   1:  PR[GP1:91,2] = PR[GP1:90,2] + 93.365;
   1:L PR[91] 10mm/sec FINE;
   1:  PR[GP1:91,1] = PR[GP1:90,1] + 106.411;
   1:  PR[GP1:91,2] = PR[GP1:90,2] + 92.968;
   1:L PR[91] 10mm/sec FINE;
   1:  PR[GP1:91,1] = PR[GP1:90,1] + 107.868;
   1:  PR[GP1:91,2] = PR[GP1:90,2] + 92.513;
   1:L PR[91] 10mm/sec FINE;
   1:  PR[GP1:91,1] = PR[GP1:90,1] + 110.644;
   1:  PR[GP1:91,2] = PR[GP1:90,2] + 92.029;
   1:L PR[91] 10mm/sec FINE;
   1:  PR[GP1:91,1] = PR[GP1:90,1] + 113.585;
   1:  PR[GP1:91,2] = PR[GP1:90,2] + 91.917;
   1:L PR[91] 10mm/sec FINE;
   1:  PR[GP1:91,1] = PR[GP1:90,1] + 116.531;
   1:  PR[GP1:91,2] = PR[GP1:90,2] + 92.230;
   1:L PR[91] 10mm/sec FINE;
   1:  PR[GP1:91,1] = PR[GP1:90,1] + 119.377;
   1:  PR[GP1:91,2] = PR[GP1:90,2] + 92.959;
   1:L PR[91] 10mm/sec FINE;
   1:  PR[GP1:91,1] = PR[GP1:90,1] + 121.994;
   1:  PR[GP1:91,2] = PR[GP1:90,2] + 94.064;
   1:L PR[91] 10mm/sec FINE;
   1:  PR[GP1:91,1] = PR[GP1:90,1] + 124.401;
   1:  PR[GP1:91,2] = PR[GP1:90,2] + 95.539;
   1:L PR[91] 10mm/sec FINE;
   1:  PR[GP1:91,1] = PR[GP1:90,1] + 126.542;
   1:  PR[GP1:91,2] = PR[GP1:90,2] + 97.347;
   1:L PR[91] 10mm/sec FINE;
   1:  PR[GP1:91,1] = PR[GP1:90,1] + 128.367;
   1:  PR[GP1:91,2] = PR[GP1:90,2] + 99.443;
   1:L PR[91] 10mm/sec FINE;
   1:  PR[GP1:91,1] = PR[GP1:90,1] + 129.834;
   1:  PR[GP1:91,2] = PR[GP1:90,2] + 101.778;
   1:L PR[91] 10mm/sec FINE;
   1:  PR[GP1:91,1] = PR[GP1:90,1] + 130.082;
   1:  PR[GP1:91,2] = PR[GP1:90,2] + 102.358;
   1:L PR[91] 10mm/sec FINE;
   1:  PR[GP1:91,1] = PR[GP1:90,1] + 130.881;
   1:  PR[GP1:91,2] = PR[GP1:90,2] + 104.290;
   1:L PR[91] 10mm/sec FINE;
   1:  PR[GP1:91,1] = PR[GP1:90,1] + 131.513;
   1:  PR[GP1:91,2] = PR[GP1:90,2] + 106.930;
   1:L PR[91] 10mm/sec FINE;
   1:  PR[GP1:91,1] = PR[GP1:90,1] + 131.608;
   1:  PR[GP1:91,2] = PR[GP1:90,2] + 107.870;
   1:L PR[91] 10mm/sec FINE;
   1:  PR[GP1:91,1] = PR[GP1:90,1] + 131.746;
   1:  PR[GP1:91,2] = PR[GP1:90,2] + 109.629;
   1:L PR[91] 10mm/sec FINE;
   1:  PR[GP1:91,1] = PR[GP1:90,1] + 131.403;
   1:  PR[GP1:91,2] = PR[GP1:90,2] + 113.038;
   1:L PR[91] 10mm/sec FINE;
   1:  PR[GP1:91,1] = PR[GP1:90,1] + 130.376;
   1:  PR[GP1:91,2] = PR[GP1:90,2] + 116.309;
   1:L PR[91] 10mm/sec FINE;
   1:  PR[GP1:91,1] = PR[GP1:90,1] + 128.692;
   1:  PR[GP1:91,2] = PR[GP1:90,2] + 119.314;
   1:L PR[91] 10mm/sec FINE;
   1:  PR[GP1:91,1] = PR[GP1:90,1] + 126.422;
   1:  PR[GP1:91,2] = PR[GP1:90,2] + 121.938;
   1:L PR[91] 10mm/sec FINE;
   1:  PR[GP1:91,1] = PR[GP1:90,1] + 123.656;
   1:  PR[GP1:91,2] = PR[GP1:90,2] + 124.077;
   1:L PR[91] 10mm/sec FINE;
   1:  PR[GP1:91,1] = PR[GP1:90,1] + 120.503;
   1:  PR[GP1:91,2] = PR[GP1:90,2] + 125.648;
   1:L PR[91] 10mm/sec FINE;
   1:  PR[GP1:91,1] = PR[GP1:90,1] + 117.094;
   1:  PR[GP1:91,2] = PR[GP1:90,2] + 126.591;
   1:L PR[91] 10mm/sec FINE;
   1:  PR[GP1:91,1] = PR[GP1:90,1] + 113.460;
   1:  PR[GP1:91,2] = PR[GP1:90,2] + 126.855;
   1:L PR[91] 10mm/sec FINE;
   1:  PR[GP1:91,1] = PR[GP1:90,1] + 109.815;
   1:  PR[GP1:91,2] = PR[GP1:90,2] + 126.442;
   1:L PR[91] 10mm/sec FINE;
   1:  PR[GP1:91,1] = PR[GP1:90,1] + 106.259;
   1:  PR[GP1:91,2] = PR[GP1:90,2] + 125.353;
   1:L PR[91] 10mm/sec FINE;
   1:  PR[GP1:91,1] = PR[GP1:90,1] + 102.967;
   1:  PR[GP1:91,2] = PR[GP1:90,2] + 123.644;
   1:L PR[91] 10mm/sec FINE;
   1:  PR[GP1:91,1] = PR[GP1:90,1] + 100.053;
   1:  PR[GP1:91,2] = PR[GP1:90,2] + 121.370;
   1:L PR[91] 10mm/sec FINE;
   1:  PR[GP1:91,1] = PR[GP1:90,1] + 97.658;
   1:  PR[GP1:91,2] = PR[GP1:90,2] + 118.630;
   1:L PR[91] 10mm/sec FINE;
   1:  PR[GP1:91,1] = PR[GP1:90,1] + 97.573;
   1:  PR[GP1:91,2] = PR[GP1:90,2] + 118.506;
   1:L PR[91] 10mm/sec FINE;
   1:  PR[GP1:91,1] = PR[GP1:90,1] + 96.390;
   1:  PR[GP1:91,2] = PR[GP1:90,2] + 116.490;
   1:L PR[91] 10mm/sec FINE;
   1:  PR[GP1:91,1] = PR[GP1:90,1] + 96.144;
   1:  PR[GP1:91,2] = PR[GP1:90,2] + 116.224;
   1:L PR[91] 10mm/sec FINE;
   1:  PR[GP1:91,1] = PR[GP1:90,1] + 95.665;
   1:  PR[GP1:91,2] = PR[GP1:90,2] + 115.648;
   1:L PR[91] 10mm/sec FINE;
   1:  PR[GP1:91,1] = PR[GP1:90,1] + 94.894;
   1:  PR[GP1:91,2] = PR[GP1:90,2] + 115.385;
   1:L PR[91] 10mm/sec FINE;
   1:  PR[GP1:91,1] = PR[GP1:90,1] + 94.595;
   1:  PR[GP1:91,2] = PR[GP1:90,2] + 115.322;
   1:L PR[91] 10mm/sec FINE;
   1:  PR[GP1:91,1] = PR[GP1:90,1] + 94.212;
   1:  PR[GP1:91,2] = PR[GP1:90,2] + 115.485;
   1:L PR[91] 10mm/sec FINE;
   1:  PR[GP1:91,1] = PR[GP1:90,1] + 93.542;
   1:  PR[GP1:91,2] = PR[GP1:90,2] + 115.632;
   1:L PR[91] 10mm/sec FINE;
   1:  PR[GP1:91,1] = PR[GP1:90,1] + 92.998;
   1:  PR[GP1:91,2] = PR[GP1:90,2] + 116.268;
   1:L PR[91] 10mm/sec FINE;
   1:  PR[GP1:91,1] = PR[GP1:90,1] + 92.725;
   1:  PR[GP1:91,2] = PR[GP1:90,2] + 116.535;
   1:L PR[91] 10mm/sec FINE;
   1:  PR[GP1:91,1] = PR[GP1:90,1] + 92.039;
   1:  PR[GP1:91,2] = PR[GP1:90,2] + 117.892;
   1:L PR[91] 10mm/sec FINE;
   1:  PR[GP1:91,1] = PR[GP1:90,1] + 91.114;
   1:  PR[GP1:91,2] = PR[GP1:90,2] + 119.148;
   1:L PR[91] 10mm/sec FINE;
   1:  PR[GP1:91,1] = PR[GP1:90,1] + 89.807;
   1:  PR[GP1:91,2] = PR[GP1:90,2] + 120.838;
   1:L PR[91] 10mm/sec FINE;
   1:  PR[GP1:91,1] = PR[GP1:90,1] + 89.143;
   1:  PR[GP1:91,2] = PR[GP1:90,2] + 121.442;
   1:L PR[91] 10mm/sec FINE;
   1:  PR[GP1:91,1] = PR[GP1:90,1] + 87.033;
   1:  PR[GP1:91,2] = PR[GP1:90,2] + 123.279;
   1:L PR[91] 10mm/sec FINE;
   1:  PR[GP1:91,1] = PR[GP1:90,1] + 84.036;
   1:  PR[GP1:91,2] = PR[GP1:90,2] + 125.037;
   1:L PR[91] 10mm/sec FINE;
   1:  PR[GP1:91,1] = PR[GP1:90,1] + 83.776;
   1:  PR[GP1:91,2] = PR[GP1:90,2] + 125.157;
   1:L PR[91] 10mm/sec FINE;
   1:  PR[GP1:91,1] = PR[GP1:90,1] + 80.948;
   1:  PR[GP1:91,2] = PR[GP1:90,2] + 126.151;
   1:L PR[91] 10mm/sec FINE;
   1:  PR[GP1:91,1] = PR[GP1:90,1] + 80.100;
   1:  PR[GP1:91,2] = PR[GP1:90,2] + 126.346;
   1:L PR[91] 10mm/sec FINE;
   1:  PR[GP1:91,1] = PR[GP1:90,1] + 77.624;
   1:  PR[GP1:91,2] = PR[GP1:90,2] + 126.695;
   1:L PR[91] 10mm/sec FINE;
   1:  PR[GP1:91,1] = PR[GP1:90,1] + 76.257;
   1:  PR[GP1:91,2] = PR[GP1:90,2] + 126.719;
   1:L PR[91] 10mm/sec FINE;
   1:  PR[GP1:91,1] = PR[GP1:90,1] + 74.185;
   1:  PR[GP1:91,2] = PR[GP1:90,2] + 126.597;
   1:L PR[91] 10mm/sec FINE;
   1:  PR[GP1:91,1] = PR[GP1:90,1] + 72.443;
   1:  PR[GP1:91,2] = PR[GP1:90,2] + 126.260;
   1:L PR[91] 10mm/sec FINE;
   1:  PR[GP1:91,1] = PR[GP1:90,1] + 70.778;
   1:  PR[GP1:91,2] = PR[GP1:90,2] + 125.820;
   1:L PR[91] 10mm/sec FINE;
   1:  PR[GP1:91,1] = PR[GP1:90,1] + 68.849;
   1:  PR[GP1:91,2] = PR[GP1:90,2] + 125.002;
   1:L PR[91] 10mm/sec FINE;
   1:  PR[GP1:91,1] = PR[GP1:90,1] + 67.556;
   1:  PR[GP1:91,2] = PR[GP1:90,2] + 124.364;
   1:L PR[91] 10mm/sec FINE;
   1:  PR[GP1:91,1] = PR[GP1:90,1] + 65.645;
   1:  PR[GP1:91,2] = PR[GP1:90,2] + 123.022;
   1:L PR[91] 10mm/sec FINE;
   1:  PR[GP1:91,1] = PR[GP1:90,1] + 64.673;
   1:  PR[GP1:91,2] = PR[GP1:90,2] + 122.267;
   1:L PR[91] 10mm/sec FINE;
   1:  PR[GP1:91,1] = PR[GP1:90,1] + 62.978;
   1:  PR[GP1:91,2] = PR[GP1:90,2] + 120.431;
   1:L PR[91] 10mm/sec FINE;
   1:  PR[GP1:91,1] = PR[GP1:90,1] + 62.273;
   1:  PR[GP1:91,2] = PR[GP1:90,2] + 119.605;
   1:L PR[91] 10mm/sec FINE;
   1:  PR[GP1:91,1] = PR[GP1:90,1] + 60.958;
   1:  PR[GP1:91,2] = PR[GP1:90,2] + 117.370;
   1:L PR[91] 10mm/sec FINE;
   1:  PR[GP1:91,1] = PR[GP1:90,1] + 60.473;
   1:  PR[GP1:91,2] = PR[GP1:90,2] + 116.491;
   1:L PR[91] 10mm/sec FINE;
   1:  PR[GP1:91,1] = PR[GP1:90,1] + 59.651;
   1:  PR[GP1:91,2] = PR[GP1:90,2] + 113.998;
   1:L PR[91] 10mm/sec FINE;
   1:  PR[GP1:91,1] = PR[GP1:90,1] + 59.357;
   1:  PR[GP1:91,2] = PR[GP1:90,2] + 113.064;
   1:L PR[91] 10mm/sec FINE;
   1:  PR[GP1:91,1] = PR[GP1:90,1] + 59.093;
   1:  PR[GP1:91,2] = PR[GP1:90,2] + 110.477;
   1:L PR[91] 10mm/sec FINE;
   1:  PR[GP1:91,1] = PR[GP1:90,1] + 58.933;
   1:  PR[GP1:91,2] = PR[GP1:90,2] + 109.489;
   1:L PR[91] 10mm/sec FINE;
   1:  PR[GP1:91,1] = PR[GP1:90,1] + 59.068;
   1:  PR[GP1:91,2] = PR[GP1:90,2] + 108.273;
   1:L PR[91] 10mm/sec FINE;
   1:  PR[GP1:91,1] = PR[GP1:90,1] + 59.281;
   1:  PR[GP1:91,2] = PR[GP1:90,2] + 106.982;
   1:L PR[91] 10mm/sec FINE;
   1:  PR[GP1:91,1] = PR[GP1:90,1] + 59.404;
   1:  PR[GP1:91,2] = PR[GP1:90,2] + 105.878;
   1:L PR[91] 10mm/sec FINE;
   1:  PR[GP1:91,1] = PR[GP1:90,1] + 59.777;
   1:  PR[GP1:91,2] = PR[GP1:90,2] + 104.702;
   1:L PR[91] 10mm/sec FINE;
   1:  PR[GP1:91,1] = PR[GP1:90,1] + 60.530;
   1:  PR[GP1:91,2] = PR[GP1:90,2] + 102.461;
   1:L PR[91] 10mm/sec FINE;
   1:  PR[GP1:91,1] = PR[GP1:90,1] + 61.244;
   1:  PR[GP1:91,2] = PR[GP1:90,2] + 101.193;
   1:L PR[91] 10mm/sec FINE;
   1:  PR[GP1:91,1] = PR[GP1:90,1] + 62.336;
   1:  PR[GP1:91,2] = PR[GP1:90,2] + 99.359;
   1:L PR[91] 10mm/sec FINE;
   1:  PR[GP1:91,1] = PR[GP1:90,1] + 63.483;
   1:  PR[GP1:91,2] = PR[GP1:90,2] + 98.037;
   1:L PR[91] 10mm/sec FINE;
   1:  PR[GP1:91,1] = PR[GP1:90,1] + 64.717;
   1:  PR[GP1:91,2] = PR[GP1:90,2] + 96.705;
   1:L PR[91] 10mm/sec FINE;
   1:  PR[GP1:91,1] = PR[GP1:90,1] + 66.397;
   1:  PR[GP1:91,2] = PR[GP1:90,2] + 95.413;
   1:L PR[91] 10mm/sec FINE;
   1:  PR[GP1:91,1] = PR[GP1:90,1] + 67.544;
   1:  PR[GP1:91,2] = PR[GP1:90,2] + 94.604;
   1:L PR[91] 10mm/sec FINE;
   1:  PR[GP1:91,1] = PR[GP1:90,1] + 70.520;
   1:  PR[GP1:91,2] = PR[GP1:90,2] + 93.186;
   1:  PR[GP1:91,3] = PR[GP1:90,3] + 14.900;
   1:L PR[91] 10mm/sec FINE;
   1:  PR[GP1:91,1] = PR[GP1:90,1] + 70.665;
   1:  PR[GP1:91,2] = PR[GP1:90,2] + 93.124;
   1:L PR[91] 10mm/sec FINE;
   1:  PR[GP1:91,1] = PR[GP1:90,1] + 74.193;
   1:  PR[GP1:91,2] = PR[GP1:90,2] + 92.191;
   1:L PR[91] 10mm/sec FINE;
   1:  PR[GP1:91,1] = PR[GP1:90,1] + 76.941;
   1:  PR[GP1:91,2] = PR[GP1:90,2] + 91.997;
   1:L PR[91] 10mm/sec FINE;
   1:  PR[GP1:91,1] = PR[GP1:90,1] + 77.958;
   1:  PR[GP1:91,2] = PR[GP1:90,2] + 91.958;
   1:L PR[91] 10mm/sec FINE;
   1:  PR[GP1:91,1] = PR[GP1:90,1] + 80.017;
   1:  PR[GP1:91,2] = PR[GP1:90,2] + 92.214;
   1:L PR[91] 10mm/sec FINE;
   1:  PR[GP1:91,1] = PR[GP1:90,1] + 81.716;
   1:  PR[GP1:91,2] = PR[GP1:90,2] + 92.489;
   1:L PR[91] 10mm/sec FINE;
   1:  PR[GP1:91,1] = PR[GP1:90,1] + 82.974;
   1:  PR[GP1:91,2] = PR[GP1:90,2] + 92.908;
   1:L PR[91] 10mm/sec FINE;
   1:  PR[GP1:91,1] = PR[GP1:90,1] + 85.293;
   1:  PR[GP1:91,2] = PR[GP1:90,2] + 93.785;
   1:L PR[91] 10mm/sec FINE;
   1:  PR[GP1:91,1] = PR[GP1:90,1] + 85.763;
   1:  PR[GP1:91,2] = PR[GP1:90,2] + 94.055;
   1:L PR[91] 10mm/sec FINE;
   1:  PR[GP1:91,1] = PR[GP1:90,1] + 87.717;
   1:  PR[GP1:91,2] = PR[GP1:90,2] + 95.298;
   1:L PR[91] 10mm/sec FINE;
   1:  PR[GP1:91,1] = PR[GP1:90,1] + 88.397;
   1:  PR[GP1:91,2] = PR[GP1:90,2] + 95.701;
   1:L PR[91] 10mm/sec FINE;
   1:  PR[GP1:91,1] = PR[GP1:90,1] + 88.557;
   1:  PR[GP1:91,2] = PR[GP1:90,2] + 95.813;
   1:L PR[91] 10mm/sec FINE;
   1:  PR[GP1:91,1] = PR[GP1:90,1] + 90.767;
   1:  PR[GP1:91,2] = PR[GP1:90,2] + 97.865;
   1:L PR[91] 10mm/sec FINE;
   1:  PR[GP1:91,1] = PR[GP1:90,1] + 91.387;
   1:  PR[GP1:91,2] = PR[GP1:90,2] + 98.554;
   1:L PR[91] 10mm/sec FINE;
   1:  PR[GP1:91,1] = PR[GP1:90,1] + 92.812;
   1:  PR[GP1:91,2] = PR[GP1:90,2] + 100.657;
   1:L PR[91] 10mm/sec FINE;
   1:  PR[GP1:91,1] = PR[GP1:90,1] + 93.383;
   1:  PR[GP1:91,2] = PR[GP1:90,2] + 101.249;
   1:L PR[91] 10mm/sec FINE;
   1:  PR[GP1:91,1] = PR[GP1:90,1] + 93.641;
   1:  PR[GP1:91,2] = PR[GP1:90,2] + 101.422;
   1:L PR[91] 10mm/sec FINE;
   1:  PR[GP1:91,1] = PR[GP1:90,1] + 94.275;
   1:  PR[GP1:91,2] = PR[GP1:90,2] + 101.612;
   1:L PR[91] 10mm/sec FINE;
   1:  PR[GP1:91,1] = PR[GP1:90,1] + 94.605;
   1:  PR[GP1:91,2] = PR[GP1:90,2] + 101.633;
   1:L PR[91] 10mm/sec FINE;
   1:  PR[GP1:91,1] = PR[GP1:90,1] + 95.231;
   1:  PR[GP1:91,2] = PR[GP1:90,2] + 101.437;
   1:L PR[91] 10mm/sec FINE;
   1:  PR[GP1:91,1] = PR[GP1:90,1] + 95.508;
   1:  PR[GP1:91,2] = PR[GP1:90,2] + 101.289;
   1:L PR[91] 10mm/sec FINE;
   1:  PR[GP1:91,1] = PR[GP1:90,1] + 96.060;
   1:  PR[GP1:91,2] = PR[GP1:90,2] + 100.681;
   1:L PR[91] 10mm/sec FINE;
   1:  PR[GP1:91,1] = PR[GP1:90,1] + 96.158;
   1:  PR[GP1:91,2] = PR[GP1:90,2] + 100.460;
   1:L PR[91] 10mm/sec FINE;
   1:  PR[GP1:91,1] = PR[GP1:90,1] + 96.407;
   1:  PR[GP1:91,2] = PR[GP1:90,2] + 100.056;
   1:L PR[91] 10mm/sec FINE;
   1:  PR[GP1:91,1] = PR[GP1:90,1] + 97.376;
   1:  PR[GP1:91,2] = PR[GP1:90,2] + 98.732;
   1:L PR[91] 10mm/sec FINE;
   1:  PR[GP1:91,1] = PR[GP1:90,1] + 98.317;
   1:  PR[GP1:91,2] = PR[GP1:90,2] + 97.605;
   1:L PR[91] 10mm/sec FINE;
   1:  PR[GP1:91,1] = PR[GP1:90,1] + 99.415;
   1:  PR[GP1:91,2] = PR[GP1:90,2] + 96.557;
   1:L PR[91] 10mm/sec FINE;
   1:  PR[GP1:91,1] = PR[GP1:90,1] + 100.269;
   1:  PR[GP1:91,2] = PR[GP1:90,2] + 95.816;
   1:L PR[91] 10mm/sec FINE;
   1:  PR[GP1:91,1] = PR[GP1:90,1] + 101.945;
   1:  PR[GP1:91,2] = PR[GP1:90,2] + 94.671;
   1:L PR[91] 10mm/sec FINE;
   1:  PR[GP1:91,1] = PR[GP1:90,1] + 102.489;
   1:  PR[GP1:91,2] = PR[GP1:90,2] + 94.332;
   1:L PR[91] 10mm/sec FINE;
   1:  PR[GP1:91,1] = PR[GP1:90,1] + 104.935;
   1:  PR[GP1:91,2] = PR[GP1:90,2] + 93.175;
   1:L PR[91] 10mm/sec FINE;
   1:  PR[GP1:91,1] = PR[GP1:90,1] + 107.578;
   1:  PR[GP1:91,2] = PR[GP1:90,2] + 92.350;
   1:L PR[91] 10mm/sec FINE;
   1:  PR[GP1:91,1] = PR[GP1:90,1] + 108.827;
   1:  PR[GP1:91,2] = PR[GP1:90,2] + 92.129;
   1:L PR[91] 10mm/sec FINE;
   1:  PR[GP1:91,1] = PR[GP1:90,1] + 110.348;
   1:  PR[GP1:91,2] = PR[GP1:90,2] + 91.892;
   1:L PR[91] 10mm/sec FINE;
   1:  PR[GP1:91,1] = PR[GP1:90,1] + 113.198;
   1:  PR[GP1:91,2] = PR[GP1:90,2] + 91.815;
   1:L PR[91] 10mm/sec FINE;
   1:  PR[GP1:91,1] = PR[GP1:90,1] + 116.141;
   1:  PR[GP1:91,2] = PR[GP1:90,2] + 92.132;
   1:L PR[91] 10mm/sec FINE;
   1:  PR[GP1:91,1] = PR[GP1:90,1] + 119.006;
   1:  PR[GP1:91,2] = PR[GP1:90,2] + 92.868;
   1:L PR[91] 10mm/sec FINE;
   1:  PR[GP1:91,1] = PR[GP1:90,1] + 121.709;
   1:  PR[GP1:91,2] = PR[GP1:90,2] + 94.002;
   1:L PR[91] 10mm/sec FINE;
   1:  PR[GP1:91,1] = PR[GP1:90,1] + 124.119;
   1:  PR[GP1:91,2] = PR[GP1:90,2] + 95.482;
   1:L PR[91] 10mm/sec FINE;
   1:  PR[GP1:91,1] = PR[GP1:90,1] + 126.262;
   1:  PR[GP1:91,2] = PR[GP1:90,2] + 97.295;
   1:L PR[91] 10mm/sec FINE;
   1:  PR[GP1:91,1] = PR[GP1:90,1] + 128.087;
   1:  PR[GP1:91,2] = PR[GP1:90,2] + 99.396;
   1:L PR[91] 10mm/sec FINE;
   1:  PR[GP1:91,1] = PR[GP1:90,1] + 129.553;
   1:  PR[GP1:91,2] = PR[GP1:90,2] + 101.737;
   1:L PR[91] 10mm/sec FINE;
   1:  PR[GP1:91,1] = PR[GP1:90,1] + 130.628;
   1:  PR[GP1:91,2] = PR[GP1:90,2] + 104.259;
   1:L PR[91] 10mm/sec FINE;
   1:  PR[GP1:91,1] = PR[GP1:90,1] + 131.284;
   1:  PR[GP1:91,2] = PR[GP1:90,2] + 106.903;
   1:L PR[91] 10mm/sec FINE;
   1:  PR[GP1:91,1] = PR[GP1:90,1] + 131.512;
   1:  PR[GP1:91,2] = PR[GP1:90,2] + 109.606;
   1:L PR[91] 10mm/sec FINE;
   1:  PR[GP1:91,1] = PR[GP1:90,1] + 131.132;
   1:  PR[GP1:91,2] = PR[GP1:90,2] + 113.012;
   1:L PR[91] 10mm/sec FINE;
   1:  PR[GP1:91,1] = PR[GP1:90,1] + 130.096;
   1:  PR[GP1:91,2] = PR[GP1:90,2] + 116.285;
   1:L PR[91] 10mm/sec FINE;
   1:  PR[GP1:91,1] = PR[GP1:90,1] + 128.408;
   1:  PR[GP1:91,2] = PR[GP1:90,2] + 119.291;
   1:L PR[91] 10mm/sec FINE;
   1:  PR[GP1:91,1] = PR[GP1:90,1] + 126.135;
   1:  PR[GP1:91,2] = PR[GP1:90,2] + 121.914;
   1:L PR[91] 10mm/sec FINE;
   1:  PR[GP1:91,1] = PR[GP1:90,1] + 123.367;
   1:  PR[GP1:91,2] = PR[GP1:90,2] + 124.053;
   1:L PR[91] 10mm/sec FINE;
   1:  PR[GP1:91,1] = PR[GP1:90,1] + 120.214;
   1:  PR[GP1:91,2] = PR[GP1:90,2] + 125.623;
   1:L PR[91] 10mm/sec FINE;
   1:  PR[GP1:91,1] = PR[GP1:90,1] + 116.723;
   1:  PR[GP1:91,2] = PR[GP1:90,2] + 126.554;
   1:L PR[91] 10mm/sec FINE;
   1:  PR[GP1:91,1] = PR[GP1:90,1] + 113.071;
   1:  PR[GP1:91,2] = PR[GP1:90,2] + 126.814;
   1:L PR[91] 10mm/sec FINE;
   1:  PR[GP1:91,1] = PR[GP1:90,1] + 110.735;
   1:  PR[GP1:91,2] = PR[GP1:90,2] + 126.549;
   1:L PR[91] 10mm/sec FINE;
   1:  PR[GP1:91,1] = PR[GP1:90,1] + 109.397;
   1:  PR[GP1:91,2] = PR[GP1:90,2] + 126.390;
   1:L PR[91] 10mm/sec FINE;
   1:  PR[GP1:91,1] = PR[GP1:90,1] + 105.817;
   1:  PR[GP1:91,2] = PR[GP1:90,2] + 125.295;
   1:L PR[91] 10mm/sec FINE;
   1:  PR[GP1:91,1] = PR[GP1:90,1] + 102.508;
   1:  PR[GP1:91,2] = PR[GP1:90,2] + 123.573;
   1:L PR[91] 10mm/sec FINE;
   1:  PR[GP1:91,1] = PR[GP1:90,1] + 99.591;
   1:  PR[GP1:91,2] = PR[GP1:90,2] + 121.302;
   1:L PR[91] 10mm/sec FINE;
   1:  PR[GP1:91,1] = PR[GP1:90,1] + 97.207;
   1:  PR[GP1:91,2] = PR[GP1:90,2] + 118.552;
   1:L PR[91] 10mm/sec FINE;
   1:  PR[GP1:91,1] = PR[GP1:90,1] + 96.820;
   1:  PR[GP1:91,2] = PR[GP1:90,2] + 117.991;
   1:L PR[91] 10mm/sec FINE;
   1:  PR[GP1:91,1] = PR[GP1:90,1] + 96.302;
   1:  PR[GP1:91,2] = PR[GP1:90,2] + 117.108;
   1:L PR[91] 10mm/sec FINE;
   1:  PR[GP1:91,1] = PR[GP1:90,1] + 95.879;
   1:  PR[GP1:91,2] = PR[GP1:90,2] + 116.651;
   1:L PR[91] 10mm/sec FINE;
   1:  PR[GP1:91,1] = PR[GP1:90,1] + 95.563;
   1:  PR[GP1:91,2] = PR[GP1:90,2] + 116.270;
   1:L PR[91] 10mm/sec FINE;
   1:  PR[GP1:91,1] = PR[GP1:90,1] + 95.048;
   1:  PR[GP1:91,2] = PR[GP1:90,2] + 116.094;
   1:L PR[91] 10mm/sec FINE;
   1:  PR[GP1:91,1] = PR[GP1:90,1] + 94.485;
   1:  PR[GP1:91,2] = PR[GP1:90,2] + 115.975;
   1:L PR[91] 10mm/sec FINE;
   1:  PR[GP1:91,1] = PR[GP1:90,1] + 93.699;
   1:  PR[GP1:91,2] = PR[GP1:90,2] + 116.310;
   1:L PR[91] 10mm/sec FINE;
   1:  PR[GP1:91,1] = PR[GP1:90,1] + 93.425;
   1:  PR[GP1:91,2] = PR[GP1:90,2] + 116.370;
   1:L PR[91] 10mm/sec FINE;
   1:  PR[GP1:91,1] = PR[GP1:90,1] + 92.649;
   1:  PR[GP1:91,2] = PR[GP1:90,2] + 117.254;
   1:L PR[91] 10mm/sec FINE;
   1:  PR[GP1:91,1] = PR[GP1:90,1] + 92.414;
   1:  PR[GP1:91,2] = PR[GP1:90,2] + 117.704;
   1:L PR[91] 10mm/sec FINE;
   1:  PR[GP1:91,1] = PR[GP1:90,1] + 90.988;
   1:  PR[GP1:91,2] = PR[GP1:90,2] + 119.641;
   1:L PR[91] 10mm/sec FINE;
   1:  PR[GP1:91,1] = PR[GP1:90,1] + 90.184;
   1:  PR[GP1:91,2] = PR[GP1:90,2] + 120.680;
   1:L PR[91] 10mm/sec FINE;
   1:  PR[GP1:91,1] = PR[GP1:90,1] + 88.950;
   1:  PR[GP1:91,2] = PR[GP1:90,2] + 121.803;
   1:L PR[91] 10mm/sec FINE;
   1:  PR[GP1:91,1] = PR[GP1:90,1] + 87.405;
   1:  PR[GP1:91,2] = PR[GP1:90,2] + 123.148;
   1:L PR[91] 10mm/sec FINE;
   1:  PR[GP1:91,1] = PR[GP1:90,1] + 86.560;
   1:  PR[GP1:91,2] = PR[GP1:90,2] + 123.657;
   1:L PR[91] 10mm/sec FINE;
   1:  PR[GP1:91,1] = PR[GP1:90,1] + 84.204;
   1:  PR[GP1:91,2] = PR[GP1:90,2] + 125.014;
   1:L PR[91] 10mm/sec FINE;
   1:  PR[GP1:91,1] = PR[GP1:90,1] + 80.822;
   1:  PR[GP1:91,2] = PR[GP1:90,2] + 126.190;
   1:L PR[91] 10mm/sec FINE;
   1:  PR[GP1:91,1] = PR[GP1:90,1] + 80.672;
   1:  PR[GP1:91,2] = PR[GP1:90,2] + 126.224;
   1:L PR[91] 10mm/sec FINE;
   1:  PR[GP1:91,1] = PR[GP1:90,1] + 77.538;
   1:  PR[GP1:91,2] = PR[GP1:90,2] + 126.665;
   1:L PR[91] 10mm/sec FINE;
   1:  PR[GP1:91,1] = PR[GP1:90,1] + 76.839;
   1:  PR[GP1:91,2] = PR[GP1:90,2] + 126.678;
   1:L PR[91] 10mm/sec FINE;
   1:  PR[GP1:91,1] = PR[GP1:90,1] + 74.147;
   1:  PR[GP1:91,2] = PR[GP1:90,2] + 126.520;
   1:L PR[91] 10mm/sec FINE;
   1:  PR[GP1:91,1] = PR[GP1:90,1] + 73.019;
   1:  PR[GP1:91,2] = PR[GP1:90,2] + 126.301;
   1:L PR[91] 10mm/sec FINE;
   1:  PR[GP1:91,1] = PR[GP1:90,1] + 70.787;
   1:  PR[GP1:91,2] = PR[GP1:90,2] + 125.712;
   1:L PR[91] 10mm/sec FINE;
   1:  PR[GP1:91,1] = PR[GP1:90,1] + 69.401;
   1:  PR[GP1:91,2] = PR[GP1:90,2] + 125.124;
   1:L PR[91] 10mm/sec FINE;
   1:  PR[GP1:91,1] = PR[GP1:90,1] + 67.609;
   1:  PR[GP1:91,2] = PR[GP1:90,2] + 124.240;
   1:L PR[91] 10mm/sec FINE;
   1:  PR[GP1:91,1] = PR[GP1:90,1] + 66.159;
   1:  PR[GP1:91,2] = PR[GP1:90,2] + 123.220;
   1:L PR[91] 10mm/sec FINE;
   1:  PR[GP1:91,1] = PR[GP1:90,1] + 64.767;
   1:  PR[GP1:91,2] = PR[GP1:90,2] + 122.140;
   1:L PR[91] 10mm/sec FINE;
   1:  PR[GP1:91,1] = PR[GP1:90,1] + 63.438;
   1:  PR[GP1:91,2] = PR[GP1:90,2] + 120.700;
   1:L PR[91] 10mm/sec FINE;
   1:  PR[GP1:91,1] = PR[GP1:90,1] + 62.401;
   1:  PR[GP1:91,2] = PR[GP1:90,2] + 119.485;
   1:L PR[91] 10mm/sec FINE;
   1:  PR[GP1:91,1] = PR[GP1:90,1] + 61.351;
   1:  PR[GP1:91,2] = PR[GP1:90,2] + 117.700;
   1:L PR[91] 10mm/sec FINE;
   1:  PR[GP1:91,1] = PR[GP1:90,1] + 60.627;
   1:  PR[GP1:91,2] = PR[GP1:90,2] + 116.387;
   1:L PR[91] 10mm/sec FINE;
   1:  PR[GP1:91,1] = PR[GP1:90,1] + 59.964;
   1:  PR[GP1:91,2] = PR[GP1:90,2] + 114.379;
   1:L PR[91] 10mm/sec FINE;
   1:  PR[GP1:91,1] = PR[GP1:90,1] + 59.525;
   1:  PR[GP1:91,2] = PR[GP1:90,2] + 112.983;
   1:L PR[91] 10mm/sec FINE;
   1:  PR[GP1:91,1] = PR[GP1:90,1] + 59.312;
   1:  PR[GP1:91,2] = PR[GP1:90,2] + 110.897;
   1:L PR[91] 10mm/sec FINE;
   1:  PR[GP1:91,1] = PR[GP1:90,1] + 59.076;
   1:  PR[GP1:91,2] = PR[GP1:90,2] + 109.446;
   1:L PR[91] 10mm/sec FINE;
   1:  PR[GP1:91,1] = PR[GP1:90,1] + 59.398;
   1:  PR[GP1:91,2] = PR[GP1:90,2] + 107.427;
   1:L PR[91] 10mm/sec FINE;
   1:  PR[GP1:91,1] = PR[GP1:90,1] + 59.575;
   1:  PR[GP1:91,2] = PR[GP1:90,2] + 105.845;
   1:L PR[91] 10mm/sec FINE;
   1:  PR[GP1:91,1] = PR[GP1:90,1] + 60.112;
   1:  PR[GP1:91,2] = PR[GP1:90,2] + 104.155;
   1:L PR[91] 10mm/sec FINE;
   1:  PR[GP1:91,1] = PR[GP1:90,1] + 60.684;
   1:  PR[GP1:91,2] = PR[GP1:90,2] + 102.451;
   1:L PR[91] 10mm/sec FINE;
   1:  PR[GP1:91,1] = PR[GP1:90,1] + 61.678;
   1:  PR[GP1:91,2] = PR[GP1:90,2] + 100.687;
   1:L PR[91] 10mm/sec FINE;
   1:  PR[GP1:91,1] = PR[GP1:90,1] + 62.463;
   1:  PR[GP1:91,2] = PR[GP1:90,2] + 99.368;
   1:L PR[91] 10mm/sec FINE;
   1:  PR[GP1:91,1] = PR[GP1:90,1] + 64.007;
   1:  PR[GP1:91,2] = PR[GP1:90,2] + 97.589;
   1:L PR[91] 10mm/sec FINE;
   1:  PR[GP1:91,1] = PR[GP1:90,1] + 64.808;
   1:  PR[GP1:91,2] = PR[GP1:90,2] + 96.726;
   1:L PR[91] 10mm/sec FINE;
   1:  PR[GP1:91,1] = PR[GP1:90,1] + 67.000;
   1:  PR[GP1:91,2] = PR[GP1:90,2] + 95.039;
   1:L PR[91] 10mm/sec FINE;
   1:  PR[GP1:91,1] = PR[GP1:90,1] + 67.587;
   1:  PR[GP1:91,2] = PR[GP1:90,2] + 94.625;
   1:L PR[91] 10mm/sec FINE;
   1:  PR[GP1:91,1] = PR[GP1:90,1] + 70.955;
   1:  PR[GP1:91,2] = PR[GP1:90,2] + 93.028;
   1:  PR[GP1:91,3] = PR[GP1:90,3] + 15.900;
   1:L PR[91] 10mm/sec FINE;
   1:  PR[GP1:91,1] = PR[GP1:90,1] + 73.576;
   1:  PR[GP1:91,2] = PR[GP1:90,2] + 92.321;
   1:L PR[91] 10mm/sec FINE;
   1:  PR[GP1:91,1] = PR[GP1:90,1] + 74.596;
   1:  PR[GP1:91,2] = PR[GP1:90,2] + 92.076;
   1:L PR[91] 10mm/sec FINE;
   1:  PR[GP1:91,1] = PR[GP1:90,1] + 76.653;
   1:  PR[GP1:91,2] = PR[GP1:90,2] + 91.931;
   1:L PR[91] 10mm/sec FINE;
   1:  PR[GP1:91,1] = PR[GP1:90,1] + 78.392;
   1:  PR[GP1:91,2] = PR[GP1:90,2] + 91.864;
   1:L PR[91] 10mm/sec FINE;
   1:  PR[GP1:91,1] = PR[GP1:90,1] + 79.698;
   1:  PR[GP1:91,2] = PR[GP1:90,2] + 92.026;
   1:L PR[91] 10mm/sec FINE;
   1:  PR[GP1:91,1] = PR[GP1:90,1] + 82.177;
   1:  PR[GP1:91,2] = PR[GP1:90,2] + 92.427;
   1:L PR[91] 10mm/sec FINE;
   1:  PR[GP1:91,1] = PR[GP1:90,1] + 82.645;
   1:  PR[GP1:91,2] = PR[GP1:90,2] + 92.583;
   1:L PR[91] 10mm/sec FINE;
   1:  PR[GP1:91,1] = PR[GP1:90,1] + 84.391;
   1:  PR[GP1:91,2] = PR[GP1:90,2] + 93.243;
   1:L PR[91] 10mm/sec FINE;
   1:  PR[GP1:91,1] = PR[GP1:90,1] + 85.547;
   1:  PR[GP1:91,2] = PR[GP1:90,2] + 93.640;
   1:L PR[91] 10mm/sec FINE;
   1:  PR[GP1:91,1] = PR[GP1:90,1] + 85.876;
   1:  PR[GP1:91,2] = PR[GP1:90,2] + 93.779;
   1:L PR[91] 10mm/sec FINE;
   1:  PR[GP1:91,1] = PR[GP1:90,1] + 88.283;
   1:  PR[GP1:91,2] = PR[GP1:90,2] + 95.204;
   1:L PR[91] 10mm/sec FINE;
   1:  PR[GP1:91,1] = PR[GP1:90,1] + 89.320;
   1:  PR[GP1:91,2] = PR[GP1:90,2] + 95.929;
   1:L PR[91] 10mm/sec FINE;
   1:  PR[GP1:91,1] = PR[GP1:90,1] + 90.721;
   1:  PR[GP1:91,2] = PR[GP1:90,2] + 97.230;
   1:L PR[91] 10mm/sec FINE;
   1:  PR[GP1:91,1] = PR[GP1:90,1] + 92.134;
   1:  PR[GP1:91,2] = PR[GP1:90,2] + 98.801;
   1:L PR[91] 10mm/sec FINE;
   1:  PR[GP1:91,1] = PR[GP1:90,1] + 92.661;
   1:  PR[GP1:91,2] = PR[GP1:90,2] + 99.574;
   1:L PR[91] 10mm/sec FINE;
   1:  PR[GP1:91,1] = PR[GP1:90,1] + 92.634;
   1:  PR[GP1:91,2] = PR[GP1:90,2] + 99.602;
   1:L PR[91] 10mm/sec FINE;
   1:  PR[GP1:91,1] = PR[GP1:90,1] + 93.469;
   1:  PR[GP1:91,2] = PR[GP1:90,2] + 100.424;
   1:L PR[91] 10mm/sec FINE;
   1:  PR[GP1:91,1] = PR[GP1:90,1] + 94.443;
   1:  PR[GP1:91,2] = PR[GP1:90,2] + 100.709;
   1:L PR[91] 10mm/sec FINE;
   1:  PR[GP1:91,1] = PR[GP1:90,1] + 95.373;
   1:  PR[GP1:91,2] = PR[GP1:90,2] + 100.415;
   1:L PR[91] 10mm/sec FINE;
   1:  PR[GP1:91,1] = PR[GP1:90,1] + 96.090;
   1:  PR[GP1:91,2] = PR[GP1:90,2] + 99.700;
   1:L PR[91] 10mm/sec FINE;
   1:  PR[GP1:91,1] = PR[GP1:90,1] + 96.627;
   1:  PR[GP1:91,2] = PR[GP1:90,2] + 98.958;
   1:L PR[91] 10mm/sec FINE;
   1:  PR[GP1:91,1] = PR[GP1:90,1] + 98.004;
   1:  PR[GP1:91,2] = PR[GP1:90,2] + 97.308;
   1:L PR[91] 10mm/sec FINE;
   1:  PR[GP1:91,1] = PR[GP1:90,1] + 98.578;
   1:  PR[GP1:91,2] = PR[GP1:90,2] + 96.761;
   1:L PR[91] 10mm/sec FINE;
   1:  PR[GP1:91,1] = PR[GP1:90,1] + 99.976;
   1:  PR[GP1:91,2] = PR[GP1:90,2] + 95.547;
   1:L PR[91] 10mm/sec FINE;
   1:  PR[GP1:91,1] = PR[GP1:90,1] + 101.012;
   1:  PR[GP1:91,2] = PR[GP1:90,2] + 94.839;
   1:L PR[91] 10mm/sec FINE;
   1:  PR[GP1:91,1] = PR[GP1:90,1] + 102.210;
   1:  PR[GP1:91,2] = PR[GP1:90,2] + 94.091;
   1:L PR[91] 10mm/sec FINE;
   1:  PR[GP1:91,1] = PR[GP1:90,1] + 103.929;
   1:  PR[GP1:91,2] = PR[GP1:90,2] + 93.279;
   1:L PR[91] 10mm/sec FINE;
   1:  PR[GP1:91,1] = PR[GP1:90,1] + 104.661;
   1:  PR[GP1:91,2] = PR[GP1:90,2] + 92.965;
   1:L PR[91] 10mm/sec FINE;
   1:  PR[GP1:91,1] = PR[GP1:90,1] + 107.285;
   1:  PR[GP1:91,2] = PR[GP1:90,2] + 92.187;
   1:L PR[91] 10mm/sec FINE;
   1:  PR[GP1:91,1] = PR[GP1:90,1] + 110.055;
   1:  PR[GP1:91,2] = PR[GP1:90,2] + 91.754;
   1:L PR[91] 10mm/sec FINE;
   1:  PR[GP1:91,1] = PR[GP1:90,1] + 111.441;
   1:  PR[GP1:91,2] = PR[GP1:90,2] + 91.715;
   1:L PR[91] 10mm/sec FINE;
   1:  PR[GP1:91,1] = PR[GP1:90,1] + 112.895;
   1:  PR[GP1:91,2] = PR[GP1:90,2] + 91.700;
   1:L PR[91] 10mm/sec FINE;
   1:  PR[GP1:91,1] = PR[GP1:90,1] + 115.753;
   1:  PR[GP1:91,2] = PR[GP1:90,2] + 92.034;
   1:L PR[91] 10mm/sec FINE;
   1:  PR[GP1:91,1] = PR[GP1:90,1] + 118.625;
   1:  PR[GP1:91,2] = PR[GP1:90,2] + 92.775;
   1:L PR[91] 10mm/sec FINE;
   1:  PR[GP1:91,1] = PR[GP1:90,1] + 121.337;
   1:  PR[GP1:91,2] = PR[GP1:90,2] + 93.914;
   1:L PR[91] 10mm/sec FINE;
   1:  PR[GP1:91,1] = PR[GP1:90,1] + 123.827;
   1:  PR[GP1:91,2] = PR[GP1:90,2] + 95.422;
   1:L PR[91] 10mm/sec FINE;
   1:  PR[GP1:91,1] = PR[GP1:90,1] + 125.981;
   1:  PR[GP1:91,2] = PR[GP1:90,2] + 97.243;
   1:L PR[91] 10mm/sec FINE;
   1:  PR[GP1:91,1] = PR[GP1:90,1] + 127.807;
   1:  PR[GP1:91,2] = PR[GP1:90,2] + 99.350;
   1:L PR[91] 10mm/sec FINE;
   1:  PR[GP1:91,1] = PR[GP1:90,1] + 129.273;
   1:  PR[GP1:91,2] = PR[GP1:90,2] + 101.695;
   1:L PR[91] 10mm/sec FINE;
   1:  PR[GP1:91,1] = PR[GP1:90,1] + 130.346;
   1:  PR[GP1:91,2] = PR[GP1:90,2] + 104.222;
   1:L PR[91] 10mm/sec FINE;
   1:  PR[GP1:91,1] = PR[GP1:90,1] + 131.000;
   1:  PR[GP1:91,2] = PR[GP1:90,2] + 106.870;
   1:L PR[91] 10mm/sec FINE;
   1:  PR[GP1:91,1] = PR[GP1:90,1] + 131.152;
   1:  PR[GP1:91,2] = PR[GP1:90,2] + 108.728;
   1:L PR[91] 10mm/sec FINE;
   1:  PR[GP1:91,1] = PR[GP1:90,1] + 131.248;
   1:  PR[GP1:91,2] = PR[GP1:90,2] + 109.582;
   1:L PR[91] 10mm/sec FINE;
   1:  PR[GP1:91,1] = PR[GP1:90,1] + 130.858;
   1:  PR[GP1:91,2] = PR[GP1:90,2] + 112.987;
   1:L PR[91] 10mm/sec FINE;
   1:  PR[GP1:91,1] = PR[GP1:90,1] + 129.816;
   1:  PR[GP1:91,2] = PR[GP1:90,2] + 116.261;
   1:L PR[91] 10mm/sec FINE;
   1:  PR[GP1:91,1] = PR[GP1:90,1] + 128.124;
   1:  PR[GP1:91,2] = PR[GP1:90,2] + 119.267;
   1:L PR[91] 10mm/sec FINE;
   1:  PR[GP1:91,1] = PR[GP1:90,1] + 125.848;
   1:  PR[GP1:91,2] = PR[GP1:90,2] + 121.891;
   1:L PR[91] 10mm/sec FINE;
   1:  PR[GP1:91,1] = PR[GP1:90,1] + 123.077;
   1:  PR[GP1:91,2] = PR[GP1:90,2] + 124.029;
   1:L PR[91] 10mm/sec FINE;
   1:  PR[GP1:91,1] = PR[GP1:90,1] + 122.188;
   1:  PR[GP1:91,2] = PR[GP1:90,2] + 124.472;
   1:L PR[91] 10mm/sec FINE;
   1:  PR[GP1:91,1] = PR[GP1:90,1] + 119.861;
   1:  PR[GP1:91,2] = PR[GP1:90,2] + 125.589;
   1:L PR[91] 10mm/sec FINE;
   1:  PR[GP1:91,1] = PR[GP1:90,1] + 116.348;
   1:  PR[GP1:91,2] = PR[GP1:90,2] + 126.516;
   1:L PR[91] 10mm/sec FINE;
   1:  PR[GP1:91,1] = PR[GP1:90,1] + 112.683;
   1:  PR[GP1:91,2] = PR[GP1:90,2] + 126.773;
   1:L PR[91] 10mm/sec FINE;
   1:  PR[GP1:91,1] = PR[GP1:90,1] + 112.361;
   1:  PR[GP1:91,2] = PR[GP1:90,2] + 126.736;
   1:L PR[91] 10mm/sec FINE;
   1:  PR[GP1:91,1] = PR[GP1:90,1] + 108.957;
   1:  PR[GP1:91,2] = PR[GP1:90,2] + 126.333;
   1:L PR[91] 10mm/sec FINE;
   1:  PR[GP1:91,1] = PR[GP1:90,1] + 105.373;
   1:  PR[GP1:91,2] = PR[GP1:90,2] + 125.234;
   1:L PR[91] 10mm/sec FINE;
   1:  PR[GP1:91,1] = PR[GP1:90,1] + 102.049;
   1:  PR[GP1:91,2] = PR[GP1:90,2] + 123.501;
   1:L PR[91] 10mm/sec FINE;
   1:  PR[GP1:91,1] = PR[GP1:90,1] + 100.467;
   1:  PR[GP1:91,2] = PR[GP1:90,2] + 122.270;
   1:L PR[91] 10mm/sec FINE;
   1:  PR[GP1:91,1] = PR[GP1:90,1] + 99.143;
   1:  PR[GP1:91,2] = PR[GP1:90,2] + 121.220;
   1:L PR[91] 10mm/sec FINE;
   1:  PR[GP1:91,1] = PR[GP1:90,1] + 96.755;
   1:  PR[GP1:91,2] = PR[GP1:90,2] + 118.475;
   1:L PR[91] 10mm/sec FINE;
   1:  PR[GP1:91,1] = PR[GP1:90,1] + 96.210;
   1:  PR[GP1:91,2] = PR[GP1:90,2] + 117.684;
   1:L PR[91] 10mm/sec FINE;
   1:  PR[GP1:91,1] = PR[GP1:90,1] + 96.024;
   1:  PR[GP1:91,2] = PR[GP1:90,2] + 117.520;
   1:L PR[91] 10mm/sec FINE;
   1:  PR[GP1:91,1] = PR[GP1:90,1] + 95.456;
   1:  PR[GP1:91,2] = PR[GP1:90,2] + 116.890;
   1:L PR[91] 10mm/sec FINE;
   1:  PR[GP1:91,1] = PR[GP1:90,1] + 95.202;
   1:  PR[GP1:91,2] = PR[GP1:90,2] + 116.803;
   1:L PR[91] 10mm/sec FINE;
   1:  PR[GP1:91,1] = PR[GP1:90,1] + 94.375;
   1:  PR[GP1:91,2] = PR[GP1:90,2] + 116.628;
   1:L PR[91] 10mm/sec FINE;
   1:  PR[GP1:91,1] = PR[GP1:90,1] + 93.679;
   1:  PR[GP1:91,2] = PR[GP1:90,2] + 116.925;
   1:L PR[91] 10mm/sec FINE;
   1:  PR[GP1:91,1] = PR[GP1:90,1] + 93.328;
   1:  PR[GP1:91,2] = PR[GP1:90,2] + 117.036;
   1:L PR[91] 10mm/sec FINE;
   1:  PR[GP1:91,1] = PR[GP1:90,1] + 92.682;
   1:  PR[GP1:91,2] = PR[GP1:90,2] + 117.724;
   1:L PR[91] 10mm/sec FINE;
   1:  PR[GP1:91,1] = PR[GP1:90,1] + 91.964;
   1:  PR[GP1:91,2] = PR[GP1:90,2] + 118.637;
   1:L PR[91] 10mm/sec FINE;
   1:  PR[GP1:91,1] = PR[GP1:90,1] + 90.559;
   1:  PR[GP1:91,2] = PR[GP1:90,2] + 120.524;
   1:L PR[91] 10mm/sec FINE;
   1:  PR[GP1:91,1] = PR[GP1:90,1] + 88.757;
   1:  PR[GP1:91,2] = PR[GP1:90,2] + 122.164;
   1:L PR[91] 10mm/sec FINE;
   1:  PR[GP1:91,1] = PR[GP1:90,1] + 87.779;
   1:  PR[GP1:91,2] = PR[GP1:90,2] + 123.016;
   1:L PR[91] 10mm/sec FINE;
   1:  PR[GP1:91,1] = PR[GP1:90,1] + 86.328;
   1:  PR[GP1:91,2] = PR[GP1:90,2] + 123.889;
   1:L PR[91] 10mm/sec FINE;
   1:  PR[GP1:91,1] = PR[GP1:90,1] + 84.569;
   1:  PR[GP1:91,2] = PR[GP1:90,2] + 124.903;
   1:L PR[91] 10mm/sec FINE;
   1:  PR[GP1:91,1] = PR[GP1:90,1] + 83.604;
   1:  PR[GP1:91,2] = PR[GP1:90,2] + 125.253;
   1:L PR[91] 10mm/sec FINE;
   1:  PR[GP1:91,1] = PR[GP1:90,1] + 81.068;
   1:  PR[GP1:91,2] = PR[GP1:90,2] + 126.123;
   1:L PR[91] 10mm/sec FINE;
   1:  PR[GP1:91,1] = PR[GP1:90,1] + 80.633;
   1:  PR[GP1:91,2] = PR[GP1:90,2] + 126.191;
   1:L PR[91] 10mm/sec FINE;
   1:  PR[GP1:91,1] = PR[GP1:90,1] + 77.460;
   1:  PR[GP1:91,2] = PR[GP1:90,2] + 126.635;
   1:L PR[91] 10mm/sec FINE;
   1:  PR[GP1:91,1] = PR[GP1:90,1] + 74.108;
   1:  PR[GP1:91,2] = PR[GP1:90,2] + 126.442;
   1:L PR[91] 10mm/sec FINE;
   1:  PR[GP1:91,1] = PR[GP1:90,1] + 73.594;
   1:  PR[GP1:91,2] = PR[GP1:90,2] + 126.342;
   1:L PR[91] 10mm/sec FINE;
   1:  PR[GP1:91,1] = PR[GP1:90,1] + 70.795;
   1:  PR[GP1:91,2] = PR[GP1:90,2] + 125.603;
   1:L PR[91] 10mm/sec FINE;
   1:  PR[GP1:91,1] = PR[GP1:90,1] + 69.953;
   1:  PR[GP1:91,2] = PR[GP1:90,2] + 125.246;
   1:L PR[91] 10mm/sec FINE;
   1:  PR[GP1:91,1] = PR[GP1:90,1] + 67.663;
   1:  PR[GP1:91,2] = PR[GP1:90,2] + 124.115;
   1:L PR[91] 10mm/sec FINE;
   1:  PR[GP1:91,1] = PR[GP1:90,1] + 66.672;
   1:  PR[GP1:91,2] = PR[GP1:90,2] + 123.419;
   1:L PR[91] 10mm/sec FINE;
   1:  PR[GP1:91,1] = PR[GP1:90,1] + 64.861;
   1:  PR[GP1:91,2] = PR[GP1:90,2] + 122.013;
   1:L PR[91] 10mm/sec FINE;
   1:  PR[GP1:91,1] = PR[GP1:90,1] + 63.897;
   1:  PR[GP1:91,2] = PR[GP1:90,2] + 120.969;
   1:L PR[91] 10mm/sec FINE;
   1:  PR[GP1:91,1] = PR[GP1:90,1] + 62.529;
   1:  PR[GP1:91,2] = PR[GP1:90,2] + 119.366;
   1:L PR[91] 10mm/sec FINE;
   1:  PR[GP1:91,1] = PR[GP1:90,1] + 61.743;
   1:  PR[GP1:91,2] = PR[GP1:90,2] + 118.030;
   1:L PR[91] 10mm/sec FINE;
   1:  PR[GP1:91,1] = PR[GP1:90,1] + 60.780;
   1:  PR[GP1:91,2] = PR[GP1:90,2] + 116.283;
   1:L PR[91] 10mm/sec FINE;
   1:  PR[GP1:91,1] = PR[GP1:90,1] + 60.277;
   1:  PR[GP1:91,2] = PR[GP1:90,2] + 114.760;
   1:L PR[91] 10mm/sec FINE;
   1:  PR[GP1:91,1] = PR[GP1:90,1] + 59.693;
   1:  PR[GP1:91,2] = PR[GP1:90,2] + 112.901;
   1:L PR[91] 10mm/sec FINE;
   1:  PR[GP1:91,1] = PR[GP1:90,1] + 59.531;
   1:  PR[GP1:91,2] = PR[GP1:90,2] + 111.317;
   1:L PR[91] 10mm/sec FINE;
   1:  PR[GP1:91,1] = PR[GP1:90,1] + 59.328;
   1:  PR[GP1:91,2] = PR[GP1:90,2] + 110.069;
   1:L PR[91] 10mm/sec FINE;
   1:  PR[GP1:91,1] = PR[GP1:90,1] + 59.266;
   1:  PR[GP1:91,2] = PR[GP1:90,2] + 109.390;
   1:L PR[91] 10mm/sec FINE;
   1:  PR[GP1:91,1] = PR[GP1:90,1] + 59.516;
   1:  PR[GP1:91,2] = PR[GP1:90,2] + 107.874;
   1:L PR[91] 10mm/sec FINE;
   1:  PR[GP1:91,1] = PR[GP1:90,1] + 59.746;
   1:  PR[GP1:91,2] = PR[GP1:90,2] + 105.811;
   1:L PR[91] 10mm/sec FINE;
   1:  PR[GP1:91,1] = PR[GP1:90,1] + 60.446;
   1:  PR[GP1:91,2] = PR[GP1:90,2] + 103.608;
   1:L PR[91] 10mm/sec FINE;
   1:  PR[GP1:91,1] = PR[GP1:90,1] + 60.838;
   1:  PR[GP1:91,2] = PR[GP1:90,2] + 102.442;
   1:L PR[91] 10mm/sec FINE;
   1:  PR[GP1:91,1] = PR[GP1:90,1] + 62.112;
   1:  PR[GP1:91,2] = PR[GP1:90,2] + 100.181;
   1:L PR[91] 10mm/sec FINE;
   1:  PR[GP1:91,1] = PR[GP1:90,1] + 62.590;
   1:  PR[GP1:91,2] = PR[GP1:90,2] + 99.377;
   1:L PR[91] 10mm/sec FINE;
   1:  PR[GP1:91,1] = PR[GP1:90,1] + 64.532;
   1:  PR[GP1:91,2] = PR[GP1:90,2] + 97.141;
   1:L PR[91] 10mm/sec FINE;
   1:  PR[GP1:91,1] = PR[GP1:90,1] + 64.898;
   1:  PR[GP1:91,2] = PR[GP1:90,2] + 96.746;
   1:L PR[91] 10mm/sec FINE;
   1:  PR[GP1:91,1] = PR[GP1:90,1] + 67.634;
   1:  PR[GP1:91,2] = PR[GP1:90,2] + 94.643;
   1:L PR[91] 10mm/sec FINE;
   1:  PR[GP1:91,1] = PR[GP1:90,1] + 70.367;
   1:  PR[GP1:91,2] = PR[GP1:90,2] + 93.347;
   1:  PR[GP1:91,3] = PR[GP1:90,3] + 16.900;
   1:L PR[91] 10mm/sec FINE;
   1:  PR[GP1:91,1] = PR[GP1:90,1] + 71.331;
   1:  PR[GP1:91,2] = PR[GP1:90,2] + 92.902;
   1:L PR[91] 10mm/sec FINE;
   1:  PR[GP1:91,1] = PR[GP1:90,1] + 73.336;
   1:  PR[GP1:91,2] = PR[GP1:90,2] + 92.362;
   1:L PR[91] 10mm/sec FINE;
   1:  PR[GP1:91,1] = PR[GP1:90,1] + 75.002;
   1:  PR[GP1:91,2] = PR[GP1:90,2] + 91.961;
   1:L PR[91] 10mm/sec FINE;
   1:  PR[GP1:91,1] = PR[GP1:90,1] + 76.366;
   1:  PR[GP1:91,2] = PR[GP1:90,2] + 91.865;
   1:L PR[91] 10mm/sec FINE;
   1:  PR[GP1:91,1] = PR[GP1:90,1] + 78.826;
   1:  PR[GP1:91,2] = PR[GP1:90,2] + 91.769;
   1:L PR[91] 10mm/sec FINE;
   1:  PR[GP1:91,1] = PR[GP1:90,1] + 79.379;
   1:  PR[GP1:91,2] = PR[GP1:90,2] + 91.838;
   1:L PR[91] 10mm/sec FINE;
   1:  PR[GP1:91,1] = PR[GP1:90,1] + 81.358;
   1:  PR[GP1:91,2] = PR[GP1:90,2] + 92.158;
   1:L PR[91] 10mm/sec FINE;
   1:  PR[GP1:91,1] = PR[GP1:90,1] + 82.419;
   1:  PR[GP1:91,2] = PR[GP1:90,2] + 92.301;
   1:L PR[91] 10mm/sec FINE;
   1:  PR[GP1:91,1] = PR[GP1:90,1] + 82.736;
   1:  PR[GP1:91,2] = PR[GP1:90,2] + 92.364;
   1:L PR[91] 10mm/sec FINE;
   1:  PR[GP1:91,1] = PR[GP1:90,1] + 85.401;
   1:  PR[GP1:91,2] = PR[GP1:90,2] + 93.279;
   1:L PR[91] 10mm/sec FINE;
   1:  PR[GP1:91,1] = PR[GP1:90,1] + 86.634;
   1:  PR[GP1:91,2] = PR[GP1:90,2] + 93.798;
   1:L PR[91] 10mm/sec FINE;
   1:  PR[GP1:91,1] = PR[GP1:90,1] + 88.169;
   1:  PR[GP1:91,2] = PR[GP1:90,2] + 94.707;
   1:L PR[91] 10mm/sec FINE;
   1:  PR[GP1:91,1] = PR[GP1:90,1] + 90.082;
   1:  PR[GP1:91,2] = PR[GP1:90,2] + 96.045;
   1:L PR[91] 10mm/sec FINE;
   1:  PR[GP1:91,1] = PR[GP1:90,1] + 90.675;
   1:  PR[GP1:91,2] = PR[GP1:90,2] + 96.595;
   1:L PR[91] 10mm/sec FINE;
   1:  PR[GP1:91,1] = PR[GP1:90,1] + 92.688;
   1:  PR[GP1:91,2] = PR[GP1:90,2] + 98.832;
   1:L PR[91] 10mm/sec FINE;
   1:  PR[GP1:91,1] = PR[GP1:90,1] + 93.399;
   1:  PR[GP1:91,2] = PR[GP1:90,2] + 99.527;
   1:L PR[91] 10mm/sec FINE;
   1:  PR[GP1:91,1] = PR[GP1:90,1] + 93.662;
   1:  PR[GP1:91,2] = PR[GP1:90,2] + 99.685;
   1:L PR[91] 10mm/sec FINE;
   1:  PR[GP1:91,1] = PR[GP1:90,1] + 94.361;
   1:  PR[GP1:91,2] = PR[GP1:90,2] + 99.878;
   1:L PR[91] 10mm/sec FINE;
   1:  PR[GP1:91,1] = PR[GP1:90,1] + 94.628;
   1:  PR[GP1:91,2] = PR[GP1:90,2] + 99.860;
   1:L PR[91] 10mm/sec FINE;
   1:  PR[GP1:91,1] = PR[GP1:90,1] + 95.332;
   1:  PR[GP1:91,2] = PR[GP1:90,2] + 99.661;
   1:L PR[91] 10mm/sec FINE;
   1:  PR[GP1:91,1] = PR[GP1:90,1] + 95.611;
   1:  PR[GP1:91,2] = PR[GP1:90,2] + 99.455;
   1:L PR[91] 10mm/sec FINE;
   1:  PR[GP1:91,1] = PR[GP1:90,1] + 95.683;
   1:  PR[GP1:91,2] = PR[GP1:90,2] + 99.354;
   1:L PR[91] 10mm/sec FINE;
   1:  PR[GP1:91,1] = PR[GP1:90,1] + 96.073;
   1:  PR[GP1:91,2] = PR[GP1:90,2] + 98.937;
   1:L PR[91] 10mm/sec FINE;
   1:  PR[GP1:91,1] = PR[GP1:90,1] + 97.688;
   1:  PR[GP1:91,2] = PR[GP1:90,2] + 97.015;
   1:L PR[91] 10mm/sec FINE;
   1:  PR[GP1:91,1] = PR[GP1:90,1] + 99.684;
   1:  PR[GP1:91,2] = PR[GP1:90,2] + 95.277;
   1:L PR[91] 10mm/sec FINE;
   1:  PR[GP1:91,1] = PR[GP1:90,1] + 100.080;
   1:  PR[GP1:91,2] = PR[GP1:90,2] + 95.007;
   1:L PR[91] 10mm/sec FINE;
   1:  PR[GP1:91,1] = PR[GP1:90,1] + 101.932;
   1:  PR[GP1:91,2] = PR[GP1:90,2] + 93.850;
   1:L PR[91] 10mm/sec FINE;
   1:  PR[GP1:91,1] = PR[GP1:90,1] + 102.898;
   1:  PR[GP1:91,2] = PR[GP1:90,2] + 93.393;
   1:L PR[91] 10mm/sec FINE;
   1:  PR[GP1:91,1] = PR[GP1:90,1] + 104.391;
   1:  PR[GP1:91,2] = PR[GP1:90,2] + 92.753;
   1:L PR[91] 10mm/sec FINE;
   1:  PR[GP1:91,1] = PR[GP1:90,1] + 106.172;
   1:  PR[GP1:91,2] = PR[GP1:90,2] + 92.225;
   1:L PR[91] 10mm/sec FINE;
   1:  PR[GP1:91,1] = PR[GP1:90,1] + 107.015;
   1:  PR[GP1:91,2] = PR[GP1:90,2] + 92.003;
   1:L PR[91] 10mm/sec FINE;
   1:  PR[GP1:91,1] = PR[GP1:90,1] + 109.759;
   1:  PR[GP1:91,2] = PR[GP1:90,2] + 91.617;
   1:L PR[91] 10mm/sec FINE;
   1:  PR[GP1:91,1] = PR[GP1:90,1] + 112.595;
   1:  PR[GP1:91,2] = PR[GP1:90,2] + 91.585;
   1:L PR[91] 10mm/sec FINE;
   1:  PR[GP1:91,1] = PR[GP1:90,1] + 114.148;
   1:  PR[GP1:91,2] = PR[GP1:90,2] + 91.767;
   1:L PR[91] 10mm/sec FINE;
   1:  PR[GP1:91,1] = PR[GP1:90,1] + 115.439;
   1:  PR[GP1:91,2] = PR[GP1:90,2] + 91.938;
   1:L PR[91] 10mm/sec FINE;
   1:  PR[GP1:91,1] = PR[GP1:90,1] + 118.243;
   1:  PR[GP1:91,2] = PR[GP1:90,2] + 92.681;
   1:L PR[91] 10mm/sec FINE;
   1:  PR[GP1:91,1] = PR[GP1:90,1] + 120.963;
   1:  PR[GP1:91,2] = PR[GP1:90,2] + 93.826;
   1:L PR[91] 10mm/sec FINE;
   1:  PR[GP1:91,1] = PR[GP1:90,1] + 123.459;
   1:  PR[GP1:91,2] = PR[GP1:90,2] + 95.340;
   1:L PR[91] 10mm/sec FINE;
   1:  PR[GP1:91,1] = PR[GP1:90,1] + 125.675;
   1:  PR[GP1:91,2] = PR[GP1:90,2] + 97.184;
   1:L PR[91] 10mm/sec FINE;
   1:  PR[GP1:91,1] = PR[GP1:90,1] + 127.527;
   1:  PR[GP1:91,2] = PR[GP1:90,2] + 99.304;
   1:L PR[91] 10mm/sec FINE;
   1:  PR[GP1:91,1] = PR[GP1:90,1] + 128.992;
   1:  PR[GP1:91,2] = PR[GP1:90,2] + 101.653;
   1:L PR[91] 10mm/sec FINE;
   1:  PR[GP1:91,1] = PR[GP1:90,1] + 130.064;
   1:  PR[GP1:91,2] = PR[GP1:90,2] + 104.184;
   1:L PR[91] 10mm/sec FINE;
   1:  PR[GP1:91,1] = PR[GP1:90,1] + 130.716;
   1:  PR[GP1:91,2] = PR[GP1:90,2] + 106.837;
   1:L PR[91] 10mm/sec FINE;
   1:  PR[GP1:91,1] = PR[GP1:90,1] + 130.814;
   1:  PR[GP1:91,2] = PR[GP1:90,2] + 108.037;
   1:L PR[91] 10mm/sec FINE;
   1:  PR[GP1:91,1] = PR[GP1:90,1] + 130.978;
   1:  PR[GP1:91,2] = PR[GP1:90,2] + 109.554;
   1:L PR[91] 10mm/sec FINE;
   1:  PR[GP1:91,1] = PR[GP1:90,1] + 130.583;
   1:  PR[GP1:91,2] = PR[GP1:90,2] + 112.962;
   1:L PR[91] 10mm/sec FINE;
   1:  PR[GP1:91,1] = PR[GP1:90,1] + 129.536;
   1:  PR[GP1:91,2] = PR[GP1:90,2] + 116.237;
   1:L PR[91] 10mm/sec FINE;
   1:  PR[GP1:91,1] = PR[GP1:90,1] + 127.840;
   1:  PR[GP1:91,2] = PR[GP1:90,2] + 119.244;
   1:L PR[91] 10mm/sec FINE;
   1:  PR[GP1:91,1] = PR[GP1:90,1] + 125.561;
   1:  PR[GP1:91,2] = PR[GP1:90,2] + 121.867;
   1:L PR[91] 10mm/sec FINE;
   1:  PR[GP1:91,1] = PR[GP1:90,1] + 122.726;
   1:  PR[GP1:91,2] = PR[GP1:90,2] + 123.995;
   1:L PR[91] 10mm/sec FINE;
   1:  PR[GP1:91,1] = PR[GP1:90,1] + 119.481;
   1:  PR[GP1:91,2] = PR[GP1:90,2] + 125.552;
   1:L PR[91] 10mm/sec FINE;
   1:  PR[GP1:91,1] = PR[GP1:90,1] + 115.971;
   1:  PR[GP1:91,2] = PR[GP1:90,2] + 126.478;
   1:L PR[91] 10mm/sec FINE;
   1:  PR[GP1:91,1] = PR[GP1:90,1] + 112.247;
   1:  PR[GP1:91,2] = PR[GP1:90,2] + 126.716;
   1:L PR[91] 10mm/sec FINE;
   1:  PR[GP1:91,1] = PR[GP1:90,1] + 108.517;
   1:  PR[GP1:91,2] = PR[GP1:90,2] + 126.276;
   1:L PR[91] 10mm/sec FINE;
   1:  PR[GP1:91,1] = PR[GP1:90,1] + 104.919;
   1:  PR[GP1:91,2] = PR[GP1:90,2] + 125.157;
   1:L PR[91] 10mm/sec FINE;
   1:  PR[GP1:91,1] = PR[GP1:90,1] + 101.590;
   1:  PR[GP1:91,2] = PR[GP1:90,2] + 123.430;
   1:L PR[91] 10mm/sec FINE;
   1:  PR[GP1:91,1] = PR[GP1:90,1] + 98.696;
   1:  PR[GP1:91,2] = PR[GP1:90,2] + 121.136;
   1:L PR[91] 10mm/sec FINE;
   1:  PR[GP1:91,1] = PR[GP1:90,1] + 96.304;
   1:  PR[GP1:91,2] = PR[GP1:90,2] + 118.397;
   1:L PR[91] 10mm/sec FINE;
   1:  PR[GP1:91,1] = PR[GP1:90,1] + 96.156;
   1:  PR[GP1:91,2] = PR[GP1:90,2] + 118.183;
   1:L PR[91] 10mm/sec FINE;
   1:  PR[GP1:91,1] = PR[GP1:90,1] + 95.347;
   1:  PR[GP1:91,2] = PR[GP1:90,2] + 117.455;
   1:L PR[91] 10mm/sec FINE;
   1:  PR[GP1:91,1] = PR[GP1:90,1] + 94.269;
   1:  PR[GP1:91,2] = PR[GP1:90,2] + 117.248;
   1:L PR[91] 10mm/sec FINE;
   1:  PR[GP1:91,1] = PR[GP1:90,1] + 94.144;
   1:  PR[GP1:91,2] = PR[GP1:90,2] + 117.309;
   1:L PR[91] 10mm/sec FINE;
   1:  PR[GP1:91,1] = PR[GP1:90,1] + 93.271;
   1:  PR[GP1:91,2] = PR[GP1:90,2] + 117.585;
   1:L PR[91] 10mm/sec FINE;
   1:  PR[GP1:91,1] = PR[GP1:90,1] + 92.719;
   1:  PR[GP1:91,2] = PR[GP1:90,2] + 118.163;
   1:L PR[91] 10mm/sec FINE;
   1:  PR[GP1:91,1] = PR[GP1:90,1] + 91.031;
   1:  PR[GP1:91,2] = PR[GP1:90,2] + 120.307;
   1:L PR[91] 10mm/sec FINE;
   1:  PR[GP1:91,1] = PR[GP1:90,1] + 90.799;
   1:  PR[GP1:91,2] = PR[GP1:90,2] + 120.529;
   1:L PR[91] 10mm/sec FINE;
   1:  PR[GP1:91,1] = PR[GP1:90,1] + 90.017;
   1:  PR[GP1:91,2] = PR[GP1:90,2] + 121.203;
   1:L PR[91] 10mm/sec FINE;
   1:  PR[GP1:91,1] = PR[GP1:90,1] + 88.150;
   1:  PR[GP1:91,2] = PR[GP1:90,2] + 122.885;
   1:L PR[91] 10mm/sec FINE;
   1:  PR[GP1:91,1] = PR[GP1:90,1] + 86.097;
   1:  PR[GP1:91,2] = PR[GP1:90,2] + 124.122;
   1:L PR[91] 10mm/sec FINE;
   1:  PR[GP1:91,1] = PR[GP1:90,1] + 84.935;
   1:  PR[GP1:91,2] = PR[GP1:90,2] + 124.791;
   1:L PR[91] 10mm/sec FINE;
   1:  PR[GP1:91,1] = PR[GP1:90,1] + 83.356;
   1:  PR[GP1:91,2] = PR[GP1:90,2] + 125.363;
   1:L PR[91] 10mm/sec FINE;
   1:  PR[GP1:91,1] = PR[GP1:90,1] + 81.424;
   1:  PR[GP1:91,2] = PR[GP1:90,2] + 126.026;
   1:L PR[91] 10mm/sec FINE;
   1:  PR[GP1:91,1] = PR[GP1:90,1] + 80.390;
   1:  PR[GP1:91,2] = PR[GP1:90,2] + 126.187;
   1:L PR[91] 10mm/sec FINE;
   1:  PR[GP1:91,1] = PR[GP1:90,1] + 77.771;
   1:  PR[GP1:91,2] = PR[GP1:90,2] + 126.553;
   1:L PR[91] 10mm/sec FINE;
   1:  PR[GP1:91,1] = PR[GP1:90,1] + 74.124;
   1:  PR[GP1:91,2] = PR[GP1:90,2] + 126.364;
   1:L PR[91] 10mm/sec FINE;
   1:  PR[GP1:91,1] = PR[GP1:90,1] + 70.804;
   1:  PR[GP1:91,2] = PR[GP1:90,2] + 125.494;
   1:L PR[91] 10mm/sec FINE;
   1:  PR[GP1:91,1] = PR[GP1:90,1] + 70.505;
   1:  PR[GP1:91,2] = PR[GP1:90,2] + 125.368;
   1:L PR[91] 10mm/sec FINE;
   1:  PR[GP1:91,1] = PR[GP1:90,1] + 67.717;
   1:  PR[GP1:91,2] = PR[GP1:90,2] + 123.991;
   1:L PR[91] 10mm/sec FINE;
   1:  PR[GP1:91,1] = PR[GP1:90,1] + 67.185;
   1:  PR[GP1:91,2] = PR[GP1:90,2] + 123.617;
   1:L PR[91] 10mm/sec FINE;
   1:  PR[GP1:91,1] = PR[GP1:90,1] + 64.955;
   1:  PR[GP1:91,2] = PR[GP1:90,2] + 121.886;
   1:L PR[91] 10mm/sec FINE;
   1:  PR[GP1:91,1] = PR[GP1:90,1] + 64.356;
   1:  PR[GP1:91,2] = PR[GP1:90,2] + 121.237;
   1:L PR[91] 10mm/sec FINE;
   1:  PR[GP1:91,1] = PR[GP1:90,1] + 62.657;
   1:  PR[GP1:91,2] = PR[GP1:90,2] + 119.247;
   1:L PR[91] 10mm/sec FINE;
   1:  PR[GP1:91,1] = PR[GP1:90,1] + 62.136;
   1:  PR[GP1:91,2] = PR[GP1:90,2] + 118.361;
   1:L PR[91] 10mm/sec FINE;
   1:  PR[GP1:91,1] = PR[GP1:90,1] + 60.933;
   1:  PR[GP1:91,2] = PR[GP1:90,2] + 116.179;
   1:L PR[91] 10mm/sec FINE;
   1:  PR[GP1:91,1] = PR[GP1:90,1] + 60.591;
   1:  PR[GP1:91,2] = PR[GP1:90,2] + 115.141;
   1:L PR[91] 10mm/sec FINE;
   1:  PR[GP1:91,1] = PR[GP1:90,1] + 59.861;
   1:  PR[GP1:91,2] = PR[GP1:90,2] + 112.819;
   1:L PR[91] 10mm/sec FINE;
   1:  PR[GP1:91,1] = PR[GP1:90,1] + 59.750;
   1:  PR[GP1:91,2] = PR[GP1:90,2] + 111.737;
   1:L PR[91] 10mm/sec FINE;
   1:  PR[GP1:91,1] = PR[GP1:90,1] + 59.611;
   1:  PR[GP1:91,2] = PR[GP1:90,2] + 110.881;
   1:L PR[91] 10mm/sec FINE;
   1:  PR[GP1:91,1] = PR[GP1:90,1] + 59.469;
   1:  PR[GP1:91,2] = PR[GP1:90,2] + 109.323;
   1:L PR[91] 10mm/sec FINE;
   1:  PR[GP1:91,1] = PR[GP1:90,1] + 59.634;
   1:  PR[GP1:91,2] = PR[GP1:90,2] + 108.321;
   1:L PR[91] 10mm/sec FINE;
   1:  PR[GP1:91,1] = PR[GP1:90,1] + 59.918;
   1:  PR[GP1:91,2] = PR[GP1:90,2] + 105.778;
   1:L PR[91] 10mm/sec FINE;
   1:  PR[GP1:91,1] = PR[GP1:90,1] + 60.781;
   1:  PR[GP1:91,2] = PR[GP1:90,2] + 103.060;
   1:L PR[91] 10mm/sec FINE;
   1:  PR[GP1:91,1] = PR[GP1:90,1] + 60.991;
   1:  PR[GP1:91,2] = PR[GP1:90,2] + 102.433;
   1:L PR[91] 10mm/sec FINE;
   1:  PR[GP1:91,1] = PR[GP1:90,1] + 62.546;
   1:  PR[GP1:91,2] = PR[GP1:90,2] + 99.675;
   1:L PR[91] 10mm/sec FINE;
   1:  PR[GP1:91,1] = PR[GP1:90,1] + 62.717;
   1:  PR[GP1:91,2] = PR[GP1:90,2] + 99.387;
   1:L PR[91] 10mm/sec FINE;
   1:  PR[GP1:91,1] = PR[GP1:90,1] + 65.020;
   1:  PR[GP1:91,2] = PR[GP1:90,2] + 96.746;
   1:L PR[91] 10mm/sec FINE;
   1:  PR[GP1:91,1] = PR[GP1:90,1] + 67.963;
   1:  PR[GP1:91,2] = PR[GP1:90,2] + 94.525;
   1:L PR[91] 10mm/sec FINE;
   1:  PR[GP1:91,1] = PR[GP1:90,1] + 70.188;
   1:  PR[GP1:91,2] = PR[GP1:90,2] + 93.478;
   1:  PR[GP1:91,3] = PR[GP1:90,3] + 17.900;
   1:L PR[91] 10mm/sec FINE;
   1:  PR[GP1:91,1] = PR[GP1:90,1] + 71.710;
   1:  PR[GP1:91,2] = PR[GP1:90,2] + 92.775;
   1:L PR[91] 10mm/sec FINE;
   1:  PR[GP1:91,1] = PR[GP1:90,1] + 73.097;
   1:  PR[GP1:91,2] = PR[GP1:90,2] + 92.402;
   1:L PR[91] 10mm/sec FINE;
   1:  PR[GP1:91,1] = PR[GP1:90,1] + 75.408;
   1:  PR[GP1:91,2] = PR[GP1:90,2] + 91.846;
   1:L PR[91] 10mm/sec FINE;
   1:  PR[GP1:91,1] = PR[GP1:90,1] + 76.079;
   1:  PR[GP1:91,2] = PR[GP1:90,2] + 91.799;
   1:L PR[91] 10mm/sec FINE;
   1:  PR[GP1:91,1] = PR[GP1:90,1] + 79.319;
   1:  PR[GP1:91,2] = PR[GP1:90,2] + 91.669;
   1:L PR[91] 10mm/sec FINE;
   1:  PR[GP1:91,1] = PR[GP1:90,1] + 82.269;
   1:  PR[GP1:91,2] = PR[GP1:90,2] + 92.066;
   1:L PR[91] 10mm/sec FINE;
   1:  PR[GP1:91,1] = PR[GP1:90,1] + 83.463;
   1:  PR[GP1:91,2] = PR[GP1:90,2] + 92.302;
   1:L PR[91] 10mm/sec FINE;
   1:  PR[GP1:91,1] = PR[GP1:90,1] + 85.255;
   1:  PR[GP1:91,2] = PR[GP1:90,2] + 92.917;
   1:L PR[91] 10mm/sec FINE;
   1:  PR[GP1:91,1] = PR[GP1:90,1] + 87.392;
   1:  PR[GP1:91,2] = PR[GP1:90,2] + 93.817;
   1:L PR[91] 10mm/sec FINE;
   1:  PR[GP1:91,1] = PR[GP1:90,1] + 88.056;
   1:  PR[GP1:91,2] = PR[GP1:90,2] + 94.210;
   1:L PR[91] 10mm/sec FINE;
   1:  PR[GP1:91,1] = PR[GP1:90,1] + 90.023;
   1:  PR[GP1:91,2] = PR[GP1:90,2] + 95.586;
   1:L PR[91] 10mm/sec FINE;
   1:  PR[GP1:91,1] = PR[GP1:90,1] + 90.695;
   1:  PR[GP1:91,2] = PR[GP1:90,2] + 96.012;
   1:L PR[91] 10mm/sec FINE;
   1:  PR[GP1:91,1] = PR[GP1:90,1] + 90.913;
   1:  PR[GP1:91,2] = PR[GP1:90,2] + 96.189;
   1:L PR[91] 10mm/sec FINE;
   1:  PR[GP1:91,1] = PR[GP1:90,1] + 92.988;
   1:  PR[GP1:91,2] = PR[GP1:90,2] + 98.309;
   1:L PR[91] 10mm/sec FINE;
   1:  PR[GP1:91,1] = PR[GP1:90,1] + 93.344;
   1:  PR[GP1:91,2] = PR[GP1:90,2] + 98.649;
   1:L PR[91] 10mm/sec FINE;
   1:  PR[GP1:91,1] = PR[GP1:90,1] + 93.833;
   1:  PR[GP1:91,2] = PR[GP1:90,2] + 98.941;
   1:L PR[91] 10mm/sec FINE;
   1:  PR[GP1:91,1] = PR[GP1:90,1] + 94.316;
   1:  PR[GP1:91,2] = PR[GP1:90,2] + 99.075;
   1:L PR[91] 10mm/sec FINE;
   1:  PR[GP1:91,1] = PR[GP1:90,1] + 94.834;
   1:  PR[GP1:91,2] = PR[GP1:90,2] + 99.039;
   1:L PR[91] 10mm/sec FINE;
   1:  PR[GP1:91,1] = PR[GP1:90,1] + 95.312;
   1:  PR[GP1:91,2] = PR[GP1:90,2] + 98.904;
   1:L PR[91] 10mm/sec FINE;
   1:  PR[GP1:91,1] = PR[GP1:90,1] + 95.821;
   1:  PR[GP1:91,2] = PR[GP1:90,2] + 98.527;
   1:L PR[91] 10mm/sec FINE;
   1:  PR[GP1:91,1] = PR[GP1:90,1] + 95.959;
   1:  PR[GP1:91,2] = PR[GP1:90,2] + 98.334;
   1:L PR[91] 10mm/sec FINE;
   1:  PR[GP1:91,1] = PR[GP1:90,1] + 96.667;
   1:  PR[GP1:91,2] = PR[GP1:90,2] + 97.510;
   1:L PR[91] 10mm/sec FINE;
   1:  PR[GP1:91,1] = PR[GP1:90,1] + 97.308;
   1:  PR[GP1:91,2] = PR[GP1:90,2] + 96.810;
   1:L PR[91] 10mm/sec FINE;
   1:  PR[GP1:91,1] = PR[GP1:90,1] + 99.397;
   1:  PR[GP1:91,2] = PR[GP1:90,2] + 95.011;
   1:L PR[91] 10mm/sec FINE;
   1:  PR[GP1:91,1] = PR[GP1:90,1] + 101.650;
   1:  PR[GP1:91,2] = PR[GP1:90,2] + 93.611;
   1:L PR[91] 10mm/sec FINE;
   1:  PR[GP1:91,1] = PR[GP1:90,1] + 104.122;
   1:  PR[GP1:91,2] = PR[GP1:90,2] + 92.540;
   1:L PR[91] 10mm/sec FINE;
   1:  PR[GP1:91,1] = PR[GP1:90,1] + 105.046;
   1:  PR[GP1:91,2] = PR[GP1:90,2] + 92.267;
   1:L PR[91] 10mm/sec FINE;
   1:  PR[GP1:91,1] = PR[GP1:90,1] + 106.749;
   1:  PR[GP1:91,2] = PR[GP1:90,2] + 91.819;
   1:L PR[91] 10mm/sec FINE;
   1:  PR[GP1:91,1] = PR[GP1:90,1] + 108.626;
   1:  PR[GP1:91,2] = PR[GP1:90,2] + 91.557;
   1:L PR[91] 10mm/sec FINE;
   1:  PR[GP1:91,1] = PR[GP1:90,1] + 109.486;
   1:  PR[GP1:91,2] = PR[GP1:90,2] + 91.460;
   1:L PR[91] 10mm/sec FINE;
   1:  PR[GP1:91,1] = PR[GP1:90,1] + 112.291;
   1:  PR[GP1:91,2] = PR[GP1:90,2] + 91.470;
   1:L PR[91] 10mm/sec FINE;
   1:  PR[GP1:91,1] = PR[GP1:90,1] + 115.128;
   1:  PR[GP1:91,2] = PR[GP1:90,2] + 91.843;
   1:L PR[91] 10mm/sec FINE;
   1:  PR[GP1:91,1] = PR[GP1:90,1] + 116.827;
   1:  PR[GP1:91,2] = PR[GP1:90,2] + 92.294;
   1:L PR[91] 10mm/sec FINE;
   1:  PR[GP1:91,1] = PR[GP1:90,1] + 117.911;
   1:  PR[GP1:91,2] = PR[GP1:90,2] + 92.599;
   1:L PR[91] 10mm/sec FINE;
   1:  PR[GP1:91,1] = PR[GP1:90,1] + 120.589;
   1:  PR[GP1:91,2] = PR[GP1:90,2] + 93.737;
   1:L PR[91] 10mm/sec FINE;
   1:  PR[GP1:91,1] = PR[GP1:90,1] + 123.091;
   1:  PR[GP1:91,2] = PR[GP1:90,2] + 95.258;
   1:L PR[91] 10mm/sec FINE;
   1:  PR[GP1:91,1] = PR[GP1:90,1] + 125.310;
   1:  PR[GP1:91,2] = PR[GP1:90,2] + 97.109;
   1:L PR[91] 10mm/sec FINE;
   1:  PR[GP1:91,1] = PR[GP1:90,1] + 127.197;
   1:  PR[GP1:91,2] = PR[GP1:90,2] + 99.245;
   1:L PR[91] 10mm/sec FINE;
   1:  PR[GP1:91,1] = PR[GP1:90,1] + 128.712;
   1:  PR[GP1:91,2] = PR[GP1:90,2] + 101.613;
   1:L PR[91] 10mm/sec FINE;
   1:  PR[GP1:91,1] = PR[GP1:90,1] + 129.781;
   1:  PR[GP1:91,2] = PR[GP1:90,2] + 104.147;
   1:L PR[91] 10mm/sec FINE;
   1:  PR[GP1:91,1] = PR[GP1:90,1] + 130.432;
   1:  PR[GP1:91,2] = PR[GP1:90,2] + 106.805;
   1:L PR[91] 10mm/sec FINE;
   1:  PR[GP1:91,1] = PR[GP1:90,1] + 130.546;
   1:  PR[GP1:91,2] = PR[GP1:90,2] + 107.970;
   1:L PR[91] 10mm/sec FINE;
   1:  PR[GP1:91,1] = PR[GP1:90,1] + 130.666;
   1:  PR[GP1:91,2] = PR[GP1:90,2] + 109.519;
   1:L PR[91] 10mm/sec FINE;
   1:  PR[GP1:91,1] = PR[GP1:90,1] + 130.307;
   1:  PR[GP1:91,2] = PR[GP1:90,2] + 112.938;
   1:L PR[91] 10mm/sec FINE;
   1:  PR[GP1:91,1] = PR[GP1:90,1] + 129.256;
   1:  PR[GP1:91,2] = PR[GP1:90,2] + 116.213;
   1:L PR[91] 10mm/sec FINE;
   1:  PR[GP1:91,1] = PR[GP1:90,1] + 128.776;
   1:  PR[GP1:91,2] = PR[GP1:90,2] + 117.063;
   1:L PR[91] 10mm/sec FINE;
   1:  PR[GP1:91,1] = PR[GP1:90,1] + 127.533;
   1:  PR[GP1:91,2] = PR[GP1:90,2] + 119.216;
   1:L PR[91] 10mm/sec FINE;
   1:  PR[GP1:91,1] = PR[GP1:90,1] + 125.196;
   1:  PR[GP1:91,2] = PR[GP1:90,2] + 121.832;
   1:L PR[91] 10mm/sec FINE;
   1:  PR[GP1:91,1] = PR[GP1:90,1] + 122.348;
   1:  PR[GP1:91,2] = PR[GP1:90,2] + 123.959;
   1:L PR[91] 10mm/sec FINE;
   1:  PR[GP1:91,1] = PR[GP1:90,1] + 119.102;
   1:  PR[GP1:91,2] = PR[GP1:90,2] + 125.514;
   1:L PR[91] 10mm/sec FINE;
   1:  PR[GP1:91,1] = PR[GP1:90,1] + 117.967;
   1:  PR[GP1:91,2] = PR[GP1:90,2] + 125.814;
   1:L PR[91] 10mm/sec FINE;
   1:  PR[GP1:91,1] = PR[GP1:90,1] + 115.536;
   1:  PR[GP1:91,2] = PR[GP1:90,2] + 126.423;
   1:L PR[91] 10mm/sec FINE;
   1:  PR[GP1:91,1] = PR[GP1:90,1] + 111.801;
   1:  PR[GP1:91,2] = PR[GP1:90,2] + 126.655;
   1:L PR[91] 10mm/sec FINE;
   1:  PR[GP1:91,1] = PR[GP1:90,1] + 109.334;
   1:  PR[GP1:91,2] = PR[GP1:90,2] + 126.365;
   1:L PR[91] 10mm/sec FINE;
   1:  PR[GP1:91,1] = PR[GP1:90,1] + 108.068;
   1:  PR[GP1:91,2] = PR[GP1:90,2] + 126.203;
   1:L PR[91] 10mm/sec FINE;
   1:  PR[GP1:91,1] = PR[GP1:90,1] + 104.466;
   1:  PR[GP1:91,2] = PR[GP1:90,2] + 125.079;
   1:L PR[91] 10mm/sec FINE;
   1:  PR[GP1:91,1] = PR[GP1:90,1] + 102.433;
   1:  PR[GP1:91,2] = PR[GP1:90,2] + 124.025;
   1:L PR[91] 10mm/sec FINE;
   1:  PR[GP1:91,1] = PR[GP1:90,1] + 101.154;
   1:  PR[GP1:91,2] = PR[GP1:90,2] + 123.341;
   1:L PR[91] 10mm/sec FINE;
   1:  PR[GP1:91,1] = PR[GP1:90,1] + 98.250;
   1:  PR[GP1:91,2] = PR[GP1:90,2] + 121.051;
   1:L PR[91] 10mm/sec FINE;
   1:  PR[GP1:91,1] = PR[GP1:90,1] + 96.807;
   1:  PR[GP1:91,2] = PR[GP1:90,2] + 119.403;
   1:L PR[91] 10mm/sec FINE;
   1:  PR[GP1:91,1] = PR[GP1:90,1] + 96.106;
   1:  PR[GP1:91,2] = PR[GP1:90,2] + 118.634;
   1:L PR[91] 10mm/sec FINE;
   1:  PR[GP1:91,1] = PR[GP1:90,1] + 95.308;
   1:  PR[GP1:91,2] = PR[GP1:90,2] + 117.902;
   1:L PR[91] 10mm/sec FINE;
   1:  PR[GP1:91,1] = PR[GP1:90,1] + 94.568;
   1:  PR[GP1:91,2] = PR[GP1:90,2] + 117.756;
   1:L PR[91] 10mm/sec FINE;
   1:  PR[GP1:91,1] = PR[GP1:90,1] + 94.216;
   1:  PR[GP1:91,2] = PR[GP1:90,2] + 117.724;
   1:L PR[91] 10mm/sec FINE;
   1:  PR[GP1:91,1] = PR[GP1:90,1] + 93.670;
   1:  PR[GP1:91,2] = PR[GP1:90,2] + 117.991;
   1:L PR[91] 10mm/sec FINE;
   1:  PR[GP1:91,1] = PR[GP1:90,1] + 93.213;
   1:  PR[GP1:91,2] = PR[GP1:90,2] + 118.135;
   1:L PR[91] 10mm/sec FINE;
   1:  PR[GP1:91,1] = PR[GP1:90,1] + 92.757;
   1:  PR[GP1:91,2] = PR[GP1:90,2] + 118.600;
   1:L PR[91] 10mm/sec FINE;
   1:  PR[GP1:91,1] = PR[GP1:90,1] + 91.658;
   1:  PR[GP1:91,2] = PR[GP1:90,2] + 119.987;
   1:L PR[91] 10mm/sec FINE;
   1:  PR[GP1:91,1] = PR[GP1:90,1] + 90.771;
   1:  PR[GP1:91,2] = PR[GP1:90,2] + 120.837;
   1:L PR[91] 10mm/sec FINE;
   1:  PR[GP1:91,1] = PR[GP1:90,1] + 88.583;
   1:  PR[GP1:91,2] = PR[GP1:90,2] + 122.725;
   1:L PR[91] 10mm/sec FINE;
   1:  PR[GP1:91,1] = PR[GP1:90,1] + 85.299;
   1:  PR[GP1:91,2] = PR[GP1:90,2] + 124.680;
   1:L PR[91] 10mm/sec FINE;
   1:  PR[GP1:91,1] = PR[GP1:90,1] + 83.109;
   1:  PR[GP1:91,2] = PR[GP1:90,2] + 125.473;
   1:L PR[91] 10mm/sec FINE;
   1:  PR[GP1:91,1] = PR[GP1:90,1] + 81.780;
   1:  PR[GP1:91,2] = PR[GP1:90,2] + 125.930;
   1:L PR[91] 10mm/sec FINE;
   1:  PR[GP1:91,1] = PR[GP1:90,1] + 80.147;
   1:  PR[GP1:91,2] = PR[GP1:90,2] + 126.183;
   1:L PR[91] 10mm/sec FINE;
   1:  PR[GP1:91,1] = PR[GP1:90,1] + 78.116;
   1:  PR[GP1:91,2] = PR[GP1:90,2] + 126.467;
   1:L PR[91] 10mm/sec FINE;
   1:  PR[GP1:91,1] = PR[GP1:90,1] + 74.456;
   1:  PR[GP1:91,2] = PR[GP1:90,2] + 126.284;
   1:L PR[91] 10mm/sec FINE;
   1:  PR[GP1:91,1] = PR[GP1:90,1] + 70.947;
   1:  PR[GP1:91,2] = PR[GP1:90,2] + 125.400;
   1:L PR[91] 10mm/sec FINE;
   1:  PR[GP1:91,1] = PR[GP1:90,1] + 68.742;
   1:  PR[GP1:91,2] = PR[GP1:90,2] + 124.347;
   1:L PR[91] 10mm/sec FINE;
   1:  PR[GP1:91,1] = PR[GP1:90,1] + 67.771;
   1:  PR[GP1:91,2] = PR[GP1:90,2] + 123.867;
   1:L PR[91] 10mm/sec FINE;
   1:  PR[GP1:91,1] = PR[GP1:90,1] + 67.698;
   1:  PR[GP1:91,2] = PR[GP1:90,2] + 123.816;
   1:L PR[91] 10mm/sec FINE;
   1:  PR[GP1:91,1] = PR[GP1:90,1] + 65.049;
   1:  PR[GP1:91,2] = PR[GP1:90,2] + 121.759;
   1:L PR[91] 10mm/sec FINE;
   1:  PR[GP1:91,1] = PR[GP1:90,1] + 64.816;
   1:  PR[GP1:91,2] = PR[GP1:90,2] + 121.506;
   1:L PR[91] 10mm/sec FINE;
   1:  PR[GP1:91,1] = PR[GP1:90,1] + 62.785;
   1:  PR[GP1:91,2] = PR[GP1:90,2] + 119.127;
   1:L PR[91] 10mm/sec FINE;
   1:  PR[GP1:91,1] = PR[GP1:90,1] + 62.528;
   1:  PR[GP1:91,2] = PR[GP1:90,2] + 118.691;
   1:L PR[91] 10mm/sec FINE;
   1:  PR[GP1:91,1] = PR[GP1:90,1] + 61.087;
   1:  PR[GP1:91,2] = PR[GP1:90,2] + 116.076;
   1:L PR[91] 10mm/sec FINE;
   1:  PR[GP1:91,1] = PR[GP1:90,1] + 60.028;
   1:  PR[GP1:91,2] = PR[GP1:90,2] + 112.737;
   1:L PR[91] 10mm/sec FINE;
   1:  PR[GP1:91,1] = PR[GP1:90,1] + 59.969;
   1:  PR[GP1:91,2] = PR[GP1:90,2] + 112.157;
   1:L PR[91] 10mm/sec FINE;
   1:  PR[GP1:91,1] = PR[GP1:90,1] + 59.894;
   1:  PR[GP1:91,2] = PR[GP1:90,2] + 111.693;
   1:L PR[91] 10mm/sec FINE;
   1:  PR[GP1:91,1] = PR[GP1:90,1] + 59.671;
   1:  PR[GP1:91,2] = PR[GP1:90,2] + 109.256;
   1:L PR[91] 10mm/sec FINE;
   1:  PR[GP1:91,1] = PR[GP1:90,1] + 59.751;
   1:  PR[GP1:91,2] = PR[GP1:90,2] + 108.767;
   1:L PR[91] 10mm/sec FINE;
   1:  PR[GP1:91,1] = PR[GP1:90,1] + 60.089;
   1:  PR[GP1:91,2] = PR[GP1:90,2] + 105.745;
   1:L PR[91] 10mm/sec FINE;
   1:  PR[GP1:91,1] = PR[GP1:90,1] + 61.146;
   1:  PR[GP1:91,2] = PR[GP1:90,2] + 102.422;
   1:L PR[91] 10mm/sec FINE;
   1:  PR[GP1:91,1] = PR[GP1:90,1] + 61.712;
   1:  PR[GP1:91,2] = PR[GP1:90,2] + 101.417;
   1:L PR[91] 10mm/sec FINE;
   1:  PR[GP1:91,1] = PR[GP1:90,1] + 62.823;
   1:  PR[GP1:91,2] = PR[GP1:90,2] + 99.507;
   1:L PR[91] 10mm/sec FINE;
   1:  PR[GP1:91,1] = PR[GP1:90,1] + 62.921;
   1:  PR[GP1:91,2] = PR[GP1:90,2] + 99.343;
   1:L PR[91] 10mm/sec FINE;
   1:  PR[GP1:91,1] = PR[GP1:90,1] + 65.354;
   1:  PR[GP1:91,2] = PR[GP1:90,2] + 96.618;
   1:L PR[91] 10mm/sec FINE;
   1:  PR[GP1:91,1] = PR[GP1:90,1] + 67.441;
   1:  PR[GP1:91,2] = PR[GP1:90,2] + 95.033;
   1:L PR[91] 10mm/sec FINE;
   1:  PR[GP1:91,1] = PR[GP1:90,1] + 68.316;
   1:  PR[GP1:91,2] = PR[GP1:90,2] + 94.395;
   1:L PR[91] 10mm/sec FINE;
   1:  PR[GP1:91,1] = PR[GP1:90,1] + 70.009;
   1:  PR[GP1:91,2] = PR[GP1:90,2] + 93.609;
   1:  PR[GP1:91,3] = PR[GP1:90,3] + 18.900;
   1:L PR[91] 10mm/sec FINE;
   1:  PR[GP1:91,1] = PR[GP1:90,1] + 72.089;
   1:  PR[GP1:91,2] = PR[GP1:90,2] + 92.649;
   1:L PR[91] 10mm/sec FINE;
   1:  PR[GP1:91,1] = PR[GP1:90,1] + 72.857;
   1:  PR[GP1:91,2] = PR[GP1:90,2] + 92.442;
   1:L PR[91] 10mm/sec FINE;
   1:  PR[GP1:91,1] = PR[GP1:90,1] + 75.811;
   1:  PR[GP1:91,2] = PR[GP1:90,2] + 91.732;
   1:L PR[91] 10mm/sec FINE;
   1:  PR[GP1:91,1] = PR[GP1:90,1] + 79.007;
   1:  PR[GP1:91,2] = PR[GP1:90,2] + 91.549;
   1:L PR[91] 10mm/sec FINE;
   1:  PR[GP1:91,1] = PR[GP1:90,1] + 79.998;
   1:  PR[GP1:91,2] = PR[GP1:90,2] + 91.545;
   1:L PR[91] 10mm/sec FINE;
   1:  PR[GP1:91,1] = PR[GP1:90,1] + 82.120;
   1:  PR[GP1:91,2] = PR[GP1:90,2] + 91.831;
   1:L PR[91] 10mm/sec FINE;
   1:  PR[GP1:91,1] = PR[GP1:90,1] + 84.191;
   1:  PR[GP1:91,2] = PR[GP1:90,2] + 92.240;
   1:L PR[91] 10mm/sec FINE;
   1:  PR[GP1:91,1] = PR[GP1:90,1] + 85.110;
   1:  PR[GP1:91,2] = PR[GP1:90,2] + 92.555;
   1:L PR[91] 10mm/sec FINE;
   1:  PR[GP1:91,1] = PR[GP1:90,1] + 87.485;
   1:  PR[GP1:91,2] = PR[GP1:90,2] + 93.556;
   1:L PR[91] 10mm/sec FINE;
   1:  PR[GP1:91,1] = PR[GP1:90,1] + 88.024;
   1:  PR[GP1:91,2] = PR[GP1:90,2] + 93.755;
   1:L PR[91] 10mm/sec FINE;
   1:  PR[GP1:91,1] = PR[GP1:90,1] + 88.234;
   1:  PR[GP1:91,2] = PR[GP1:90,2] + 93.861;
   1:L PR[91] 10mm/sec FINE;
   1:  PR[GP1:91,1] = PR[GP1:90,1] + 90.816;
   1:  PR[GP1:91,2] = PR[GP1:90,2] + 95.496;
   1:L PR[91] 10mm/sec FINE;
   1:  PR[GP1:91,1] = PR[GP1:90,1] + 91.991;
   1:  PR[GP1:91,2] = PR[GP1:90,2] + 96.450;
   1:L PR[91] 10mm/sec FINE;
   1:  PR[GP1:91,1] = PR[GP1:90,1] + 93.285;
   1:  PR[GP1:91,2] = PR[GP1:90,2] + 97.768;
   1:L PR[91] 10mm/sec FINE;
   1:  PR[GP1:91,1] = PR[GP1:90,1] + 94.005;
   1:  PR[GP1:91,2] = PR[GP1:90,2] + 98.197;
   1:L PR[91] 10mm/sec FINE;
   1:  PR[GP1:91,1] = PR[GP1:90,1] + 94.272;
   1:  PR[GP1:91,2] = PR[GP1:90,2] + 98.271;
   1:L PR[91] 10mm/sec FINE;
   1:  PR[GP1:91,1] = PR[GP1:90,1] + 95.040;
   1:  PR[GP1:91,2] = PR[GP1:90,2] + 98.218;
   1:L PR[91] 10mm/sec FINE;
   1:  PR[GP1:91,1] = PR[GP1:90,1] + 95.292;
   1:  PR[GP1:91,2] = PR[GP1:90,2] + 98.147;
   1:L PR[91] 10mm/sec FINE;
   1:  PR[GP1:91,1] = PR[GP1:90,1] + 96.032;
   1:  PR[GP1:91,2] = PR[GP1:90,2] + 97.599;
   1:L PR[91] 10mm/sec FINE;
   1:  PR[GP1:91,1] = PR[GP1:90,1] + 96.123;
   1:  PR[GP1:91,2] = PR[GP1:90,2] + 97.472;
   1:L PR[91] 10mm/sec FINE;
   1:  PR[GP1:91,1] = PR[GP1:90,1] + 96.453;
   1:  PR[GP1:91,2] = PR[GP1:90,2] + 97.102;
   1:L PR[91] 10mm/sec FINE;
   1:  PR[GP1:91,1] = PR[GP1:90,1] + 96.922;
   1:  PR[GP1:91,2] = PR[GP1:90,2] + 96.615;
   1:L PR[91] 10mm/sec FINE;
   1:  PR[GP1:91,1] = PR[GP1:90,1] + 98.439;
   1:  PR[GP1:91,2] = PR[GP1:90,2] + 95.292;
   1:L PR[91] 10mm/sec FINE;
   1:  PR[GP1:91,1] = PR[GP1:90,1] + 99.126;
   1:  PR[GP1:91,2] = PR[GP1:90,2] + 94.743;
   1:L PR[91] 10mm/sec FINE;
   1:  PR[GP1:91,1] = PR[GP1:90,1] + 100.978;
   1:  PR[GP1:91,2] = PR[GP1:90,2] + 93.599;
   1:L PR[91] 10mm/sec FINE;
   1:  PR[GP1:91,1] = PR[GP1:90,1] + 101.384;
   1:  PR[GP1:91,2] = PR[GP1:90,2] + 93.367;
   1:L PR[91] 10mm/sec FINE;
   1:  PR[GP1:91,1] = PR[GP1:90,1] + 103.849;
   1:  PR[GP1:91,2] = PR[GP1:90,2] + 92.329;
   1:L PR[91] 10mm/sec FINE;
   1:  PR[GP1:91,1] = PR[GP1:90,1] + 106.483;
   1:  PR[GP1:91,2] = PR[GP1:90,2] + 91.634;
   1:L PR[91] 10mm/sec FINE;
   1:  PR[GP1:91,1] = PR[GP1:90,1] + 107.412;
   1:  PR[GP1:91,2] = PR[GP1:90,2] + 91.504;
   1:L PR[91] 10mm/sec FINE;
   1:  PR[GP1:91,1] = PR[GP1:90,1] + 109.218;
   1:  PR[GP1:91,2] = PR[GP1:90,2] + 91.302;
   1:L PR[91] 10mm/sec FINE;
   1:  PR[GP1:91,1] = PR[GP1:90,1] + 111.225;
   1:  PR[GP1:91,2] = PR[GP1:90,2] + 91.316;
   1:L PR[91] 10mm/sec FINE;
   1:  PR[GP1:91,1] = PR[GP1:90,1] + 112.008;
   1:  PR[GP1:91,2] = PR[GP1:90,2] + 91.339;
   1:L PR[91] 10mm/sec FINE;
   1:  PR[GP1:91,1] = PR[GP1:90,1] + 113.888;
   1:  PR[GP1:91,2] = PR[GP1:90,2] + 91.624;
   1:L PR[91] 10mm/sec FINE;
   1:  PR[GP1:91,1] = PR[GP1:90,1] + 114.816;
   1:  PR[GP1:91,2] = PR[GP1:90,2] + 91.747;
   1:L PR[91] 10mm/sec FINE;
   1:  PR[GP1:91,1] = PR[GP1:90,1] + 117.587;
   1:  PR[GP1:91,2] = PR[GP1:90,2] + 92.519;
   1:L PR[91] 10mm/sec FINE;
   1:  PR[GP1:91,1] = PR[GP1:90,1] + 119.353;
   1:  PR[GP1:91,2] = PR[GP1:90,2] + 93.272;
   1:L PR[91] 10mm/sec FINE;
   1:  PR[GP1:91,1] = PR[GP1:90,1] + 120.242;
   1:  PR[GP1:91,2] = PR[GP1:90,2] + 93.665;
   1:L PR[91] 10mm/sec FINE;
   1:  PR[GP1:91,1] = PR[GP1:90,1] + 122.722;
   1:  PR[GP1:91,2] = PR[GP1:90,2] + 95.176;
   1:L PR[91] 10mm/sec FINE;
   1:  PR[GP1:91,1] = PR[GP1:90,1] + 124.945;
   1:  PR[GP1:91,2] = PR[GP1:90,2] + 97.034;
   1:L PR[91] 10mm/sec FINE;
   1:  PR[GP1:91,1] = PR[GP1:90,1] + 126.834;
   1:  PR[GP1:91,2] = PR[GP1:90,2] + 99.176;
   1:L PR[91] 10mm/sec FINE;
   1:  PR[GP1:91,1] = PR[GP1:90,1] + 128.348;
   1:  PR[GP1:91,2] = PR[GP1:90,2] + 101.551;
   1:L PR[91] 10mm/sec FINE;
   1:  PR[GP1:91,1] = PR[GP1:90,1] + 129.457;
   1:  PR[GP1:91,2] = PR[GP1:90,2] + 104.102;
   1:L PR[91] 10mm/sec FINE;
   1:  PR[GP1:91,1] = PR[GP1:90,1] + 130.134;
   1:  PR[GP1:91,2] = PR[GP1:90,2] + 106.769;
   1:L PR[91] 10mm/sec FINE;
   1:  PR[GP1:91,1] = PR[GP1:90,1] + 130.354;
   1:  PR[GP1:91,2] = PR[GP1:90,2] + 109.486;
   1:L PR[91] 10mm/sec FINE;
   1:  PR[GP1:91,1] = PR[GP1:90,1] + 129.967;
   1:  PR[GP1:91,2] = PR[GP1:90,2] + 112.902;
   1:L PR[91] 10mm/sec FINE;
   1:  PR[GP1:91,1] = PR[GP1:90,1] + 128.900;
   1:  PR[GP1:91,2] = PR[GP1:90,2] + 116.177;
   1:L PR[91] 10mm/sec FINE;
   1:  PR[GP1:91,1] = PR[GP1:90,1] + 127.162;
   1:  PR[GP1:91,2] = PR[GP1:90,2] + 119.180;
   1:L PR[91] 10mm/sec FINE;
   1:  PR[GP1:91,1] = PR[GP1:90,1] + 124.820;
   1:  PR[GP1:91,2] = PR[GP1:90,2] + 121.796;
   1:L PR[91] 10mm/sec FINE;
   1:  PR[GP1:91,1] = PR[GP1:90,1] + 121.969;
   1:  PR[GP1:91,2] = PR[GP1:90,2] + 123.923;
   1:L PR[91] 10mm/sec FINE;
   1:  PR[GP1:91,1] = PR[GP1:90,1] + 120.039;
   1:  PR[GP1:91,2] = PR[GP1:90,2] + 124.847;
   1:L PR[91] 10mm/sec FINE;
   1:  PR[GP1:91,1] = PR[GP1:90,1] + 118.695;
   1:  PR[GP1:91,2] = PR[GP1:90,2] + 125.467;
   1:L PR[91] 10mm/sec FINE;
   1:  PR[GP1:91,1] = PR[GP1:90,1] + 115.099;
   1:  PR[GP1:91,2] = PR[GP1:90,2] + 126.368;
   1:L PR[91] 10mm/sec FINE;
   1:  PR[GP1:91,1] = PR[GP1:90,1] + 111.355;
   1:  PR[GP1:91,2] = PR[GP1:90,2] + 126.595;
   1:L PR[91] 10mm/sec FINE;
   1:  PR[GP1:91,1] = PR[GP1:90,1] + 110.575;
   1:  PR[GP1:91,2] = PR[GP1:90,2] + 126.503;
   1:L PR[91] 10mm/sec FINE;
   1:  PR[GP1:91,1] = PR[GP1:90,1] + 107.616;
   1:  PR[GP1:91,2] = PR[GP1:90,2] + 126.125;
   1:L PR[91] 10mm/sec FINE;
   1:  PR[GP1:91,1] = PR[GP1:90,1] + 104.013;
   1:  PR[GP1:91,2] = PR[GP1:90,2] + 125.002;
   1:L PR[91] 10mm/sec FINE;
   1:  PR[GP1:91,1] = PR[GP1:90,1] + 100.717;
   1:  PR[GP1:91,2] = PR[GP1:90,2] + 123.251;
   1:L PR[91] 10mm/sec FINE;
   1:  PR[GP1:91,1] = PR[GP1:90,1] + 97.803;
   1:  PR[GP1:91,2] = PR[GP1:90,2] + 120.964;
   1:L PR[91] 10mm/sec FINE;
   1:  PR[GP1:91,1] = PR[GP1:90,1] + 96.073;
   1:  PR[GP1:91,2] = PR[GP1:90,2] + 119.064;
   1:L PR[91] 10mm/sec FINE;
   1:  PR[GP1:91,1] = PR[GP1:90,1] + 95.698;
   1:  PR[GP1:91,2] = PR[GP1:90,2] + 118.748;
   1:L PR[91] 10mm/sec FINE;
   1:  PR[GP1:91,1] = PR[GP1:90,1] + 95.268;
   1:  PR[GP1:91,2] = PR[GP1:90,2] + 118.348;
   1:L PR[91] 10mm/sec FINE;
   1:  PR[GP1:91,1] = PR[GP1:90,1] + 94.766;
   1:  PR[GP1:91,2] = PR[GP1:90,2] + 118.249;
   1:L PR[91] 10mm/sec FINE;
   1:  PR[GP1:91,1] = PR[GP1:90,1] + 94.172;
   1:  PR[GP1:91,2] = PR[GP1:90,2] + 118.195;
   1:L PR[91] 10mm/sec FINE;
   1:  PR[GP1:91,1] = PR[GP1:90,1] + 93.146;
   1:  PR[GP1:91,2] = PR[GP1:90,2] + 118.695;
   1:L PR[91] 10mm/sec FINE;
   1:  PR[GP1:91,1] = PR[GP1:90,1] + 92.797;
   1:  PR[GP1:91,2] = PR[GP1:90,2] + 119.036;
   1:L PR[91] 10mm/sec FINE;
   1:  PR[GP1:91,1] = PR[GP1:90,1] + 92.286;
   1:  PR[GP1:91,2] = PR[GP1:90,2] + 119.667;
   1:L PR[91] 10mm/sec FINE;
   1:  PR[GP1:91,1] = PR[GP1:90,1] + 90.743;
   1:  PR[GP1:91,2] = PR[GP1:90,2] + 121.146;
   1:L PR[91] 10mm/sec FINE;
   1:  PR[GP1:91,1] = PR[GP1:90,1] + 89.187;
   1:  PR[GP1:91,2] = PR[GP1:90,2] + 122.489;
   1:L PR[91] 10mm/sec FINE;
   1:  PR[GP1:91,1] = PR[GP1:90,1] + 88.358;
   1:  PR[GP1:91,2] = PR[GP1:90,2] + 123.017;
   1:L PR[91] 10mm/sec FINE;
   1:  PR[GP1:91,1] = PR[GP1:90,1] + 85.672;
   1:  PR[GP1:91,2] = PR[GP1:90,2] + 124.566;
   1:L PR[91] 10mm/sec FINE;
   1:  PR[GP1:91,1] = PR[GP1:90,1] + 82.863;
   1:  PR[GP1:91,2] = PR[GP1:90,2] + 125.583;
   1:L PR[91] 10mm/sec FINE;
   1:  PR[GP1:91,1] = PR[GP1:90,1] + 82.135;
   1:  PR[GP1:91,2] = PR[GP1:90,2] + 125.833;
   1:L PR[91] 10mm/sec FINE;
   1:  PR[GP1:91,1] = PR[GP1:90,1] + 79.903;
   1:  PR[GP1:91,2] = PR[GP1:90,2] + 126.179;
   1:L PR[91] 10mm/sec FINE;
   1:  PR[GP1:91,1] = PR[GP1:90,1] + 78.459;
   1:  PR[GP1:91,2] = PR[GP1:90,2] + 126.381;
   1:L PR[91] 10mm/sec FINE;
   1:  PR[GP1:91,1] = PR[GP1:90,1] + 76.818;
   1:  PR[GP1:91,2] = PR[GP1:90,2] + 126.313;
   1:L PR[91] 10mm/sec FINE;
   1:  PR[GP1:91,1] = PR[GP1:90,1] + 74.790;
   1:  PR[GP1:91,2] = PR[GP1:90,2] + 126.204;
   1:L PR[91] 10mm/sec FINE;
   1:  PR[GP1:91,1] = PR[GP1:90,1] + 71.270;
   1:  PR[GP1:91,2] = PR[GP1:90,2] + 125.323;
   1:L PR[91] 10mm/sec FINE;
   1:  PR[GP1:91,1] = PR[GP1:90,1] + 68.036;
   1:  PR[GP1:91,2] = PR[GP1:90,2] + 123.782;
   1:L PR[91] 10mm/sec FINE;
   1:  PR[GP1:91,1] = PR[GP1:90,1] + 67.728;
   1:  PR[GP1:91,2] = PR[GP1:90,2] + 123.552;
   1:L PR[91] 10mm/sec FINE;
   1:  PR[GP1:91,1] = PR[GP1:90,1] + 65.213;
   1:  PR[GP1:91,2] = PR[GP1:90,2] + 121.649;
   1:L PR[91] 10mm/sec FINE;
   1:  PR[GP1:91,1] = PR[GP1:90,1] + 62.914;
   1:  PR[GP1:91,2] = PR[GP1:90,2] + 119.009;
   1:L PR[91] 10mm/sec FINE;
   1:  PR[GP1:91,1] = PR[GP1:90,1] + 61.240;
   1:  PR[GP1:91,2] = PR[GP1:90,2] + 115.973;
   1:L PR[91] 10mm/sec FINE;
   1:  PR[GP1:91,1] = PR[GP1:90,1] + 60.196;
   1:  PR[GP1:91,2] = PR[GP1:90,2] + 112.656;
   1:L PR[91] 10mm/sec FINE;
   1:  PR[GP1:91,1] = PR[GP1:90,1] + 59.874;
   1:  PR[GP1:91,2] = PR[GP1:90,2] + 109.189;
   1:L PR[91] 10mm/sec FINE;
   1:  PR[GP1:91,1] = PR[GP1:90,1] + 60.301;
   1:  PR[GP1:91,2] = PR[GP1:90,2] + 105.689;
   1:L PR[91] 10mm/sec FINE;
   1:  PR[GP1:91,1] = PR[GP1:90,1] + 61.420;
   1:  PR[GP1:91,2] = PR[GP1:90,2] + 102.330;
   1:L PR[91] 10mm/sec FINE;
   1:  PR[GP1:91,1] = PR[GP1:90,1] + 62.874;
   1:  PR[GP1:91,2] = PR[GP1:90,2] + 99.829;
   1:L PR[91] 10mm/sec FINE;
   1:  PR[GP1:91,1] = PR[GP1:90,1] + 63.240;
   1:  PR[GP1:91,2] = PR[GP1:90,2] + 99.219;
   1:L PR[91] 10mm/sec FINE;
   1:  PR[GP1:91,1] = PR[GP1:90,1] + 64.920;
   1:  PR[GP1:91,2] = PR[GP1:90,2] + 97.326;
   1:L PR[91] 10mm/sec FINE;
   1:  PR[GP1:91,1] = PR[GP1:90,1] + 65.688;
   1:  PR[GP1:91,2] = PR[GP1:90,2] + 96.489;
   1:L PR[91] 10mm/sec FINE;
   1:  PR[GP1:91,1] = PR[GP1:90,1] + 67.331;
   1:  PR[GP1:91,2] = PR[GP1:90,2] + 95.241;
   1:L PR[91] 10mm/sec FINE;
   1:  PR[GP1:91,1] = PR[GP1:90,1] + 68.671;
   1:  PR[GP1:91,2] = PR[GP1:90,2] + 94.264;
   1:L PR[91] 10mm/sec FINE;
   1:  PR[GP1:91,1] = PR[GP1:90,1] + 69.829;
   1:  PR[GP1:91,2] = PR[GP1:90,2] + 93.740;
   1:  PR[GP1:91,3] = PR[GP1:90,3] + 19.900;
   1:L PR[91] 10mm/sec FINE;
   1:  PR[GP1:91,1] = PR[GP1:90,1] + 72.465;
   1:  PR[GP1:91,2] = PR[GP1:90,2] + 92.523;
   1:L PR[91] 10mm/sec FINE;
   1:  PR[GP1:91,1] = PR[GP1:90,1] + 75.728;
   1:  PR[GP1:91,2] = PR[GP1:90,2] + 91.712;
   1:L PR[91] 10mm/sec FINE;
   1:  PR[GP1:91,1] = PR[GP1:90,1] + 76.440;
   1:  PR[GP1:91,2] = PR[GP1:90,2] + 91.568;
   1:L PR[91] 10mm/sec FINE;
   1:  PR[GP1:91,1] = PR[GP1:90,1] + 78.875;
   1:  PR[GP1:91,2] = PR[GP1:90,2] + 91.429;
   1:L PR[91] 10mm/sec FINE;
   1:  PR[GP1:91,1] = PR[GP1:90,1] + 80.680;
   1:  PR[GP1:91,2] = PR[GP1:90,2] + 91.422;
   1:L PR[91] 10mm/sec FINE;
   1:  PR[GP1:91,1] = PR[GP1:90,1] + 81.970;
   1:  PR[GP1:91,2] = PR[GP1:90,2] + 91.596;
   1:L PR[91] 10mm/sec FINE;
   1:  PR[GP1:91,1] = PR[GP1:90,1] + 84.916;
   1:  PR[GP1:91,2] = PR[GP1:90,2] + 92.177;
   1:L PR[91] 10mm/sec FINE;
   1:  PR[GP1:91,1] = PR[GP1:90,1] + 88.159;
   1:  PR[GP1:91,2] = PR[GP1:90,2] + 93.378;
   1:L PR[91] 10mm/sec FINE;
   1:  PR[GP1:91,1] = PR[GP1:90,1] + 89.414;
   1:  PR[GP1:91,2] = PR[GP1:90,2] + 94.016;
   1:L PR[91] 10mm/sec FINE;
   1:  PR[GP1:91,1] = PR[GP1:90,1] + 90.937;
   1:  PR[GP1:91,2] = PR[GP1:90,2] + 94.980;
   1:L PR[91] 10mm/sec FINE;
   1:  PR[GP1:91,1] = PR[GP1:90,1] + 93.068;
   1:  PR[GP1:91,2] = PR[GP1:90,2] + 96.712;
   1:L PR[91] 10mm/sec FINE;
   1:  PR[GP1:91,1] = PR[GP1:90,1] + 93.312;
   1:  PR[GP1:91,2] = PR[GP1:90,2] + 96.964;
   1:L PR[91] 10mm/sec FINE;
   1:  PR[GP1:91,1] = PR[GP1:90,1] + 94.208;
   1:  PR[GP1:91,2] = PR[GP1:90,2] + 97.473;
   1:L PR[91] 10mm/sec FINE;
   1:  PR[GP1:91,1] = PR[GP1:90,1] + 95.278;
   1:  PR[GP1:91,2] = PR[GP1:90,2] + 97.411;
   1:L PR[91] 10mm/sec FINE;
   1:  PR[GP1:91,1] = PR[GP1:90,1] + 96.161;
   1:  PR[GP1:91,2] = PR[GP1:90,2] + 96.810;
   1:L PR[91] 10mm/sec FINE;
   1:  PR[GP1:91,1] = PR[GP1:90,1] + 96.538;
   1:  PR[GP1:91,2] = PR[GP1:90,2] + 96.419;
   1:L PR[91] 10mm/sec FINE;
   1:  PR[GP1:91,1] = PR[GP1:90,1] + 97.657;
   1:  PR[GP1:91,2] = PR[GP1:90,2] + 95.432;
   1:L PR[91] 10mm/sec FINE;
   1:  PR[GP1:91,1] = PR[GP1:90,1] + 98.860;
   1:  PR[GP1:91,2] = PR[GP1:90,2] + 94.474;
   1:L PR[91] 10mm/sec FINE;
   1:  PR[GP1:91,1] = PR[GP1:90,1] + 100.120;
   1:  PR[GP1:91,2] = PR[GP1:90,2] + 93.694;
   1:L PR[91] 10mm/sec FINE;
   1:  PR[GP1:91,1] = PR[GP1:90,1] + 101.128;
   1:  PR[GP1:91,2] = PR[GP1:90,2] + 93.120;
   1:L PR[91] 10mm/sec FINE;
   1:  PR[GP1:91,1] = PR[GP1:90,1] + 102.974;
   1:  PR[GP1:91,2] = PR[GP1:90,2] + 92.345;
   1:L PR[91] 10mm/sec FINE;
   1:  PR[GP1:91,1] = PR[GP1:90,1] + 103.596;
   1:  PR[GP1:91,2] = PR[GP1:90,2] + 92.106;
   1:L PR[91] 10mm/sec FINE;
   1:  PR[GP1:91,1] = PR[GP1:90,1] + 106.209;
   1:  PR[GP1:91,2] = PR[GP1:90,2] + 91.451;
   1:L PR[91] 10mm/sec FINE;
   1:  PR[GP1:91,1] = PR[GP1:90,1] + 108.951;
   1:  PR[GP1:91,2] = PR[GP1:90,2] + 91.143;
   1:L PR[91] 10mm/sec FINE;
   1:  PR[GP1:91,1] = PR[GP1:90,1] + 109.938;
   1:  PR[GP1:91,2] = PR[GP1:90,2] + 91.150;
   1:L PR[91] 10mm/sec FINE;
   1:  PR[GP1:91,1] = PR[GP1:90,1] + 111.734;
   1:  PR[GP1:91,2] = PR[GP1:90,2] + 91.205;
   1:L PR[91] 10mm/sec FINE;
   1:  PR[GP1:91,1] = PR[GP1:90,1] + 113.882;
   1:  PR[GP1:91,2] = PR[GP1:90,2] + 91.530;
   1:L PR[91] 10mm/sec FINE;
   1:  PR[GP1:91,1] = PR[GP1:90,1] + 114.516;
   1:  PR[GP1:91,2] = PR[GP1:90,2] + 91.639;
   1:L PR[91] 10mm/sec FINE;
   1:  PR[GP1:91,1] = PR[GP1:90,1] + 115.940;
   1:  PR[GP1:91,2] = PR[GP1:90,2] + 92.068;
   1:L PR[91] 10mm/sec FINE;
   1:  PR[GP1:91,1] = PR[GP1:90,1] + 117.262;
   1:  PR[GP1:91,2] = PR[GP1:90,2] + 92.439;
   1:L PR[91] 10mm/sec FINE;
   1:  PR[GP1:91,1] = PR[GP1:90,1] + 119.903;
   1:  PR[GP1:91,2] = PR[GP1:90,2] + 93.597;
   1:L PR[91] 10mm/sec FINE;
   1:  PR[GP1:91,1] = PR[GP1:90,1] + 121.621;
   1:  PR[GP1:91,2] = PR[GP1:90,2] + 94.645;
   1:L PR[91] 10mm/sec FINE;
   1:  PR[GP1:91,1] = PR[GP1:90,1] + 122.363;
   1:  PR[GP1:91,2] = PR[GP1:90,2] + 95.110;
   1:L PR[91] 10mm/sec FINE;
   1:  PR[GP1:91,1] = PR[GP1:90,1] + 124.579;
   1:  PR[GP1:91,2] = PR[GP1:90,2] + 96.958;
   1:L PR[91] 10mm/sec FINE;
   1:  PR[GP1:91,1] = PR[GP1:90,1] + 126.470;
   1:  PR[GP1:91,2] = PR[GP1:90,2] + 99.107;
   1:L PR[91] 10mm/sec FINE;
   1:  PR[GP1:91,1] = PR[GP1:90,1] + 127.984;
   1:  PR[GP1:91,2] = PR[GP1:90,2] + 101.489;
   1:L PR[91] 10mm/sec FINE;
   1:  PR[GP1:91,1] = PR[GP1:90,1] + 129.092;
   1:  PR[GP1:91,2] = PR[GP1:90,2] + 104.046;
   1:L PR[91] 10mm/sec FINE;
   1:  PR[GP1:91,1] = PR[GP1:90,1] + 129.767;
   1:  PR[GP1:91,2] = PR[GP1:90,2] + 106.718;
   1:L PR[91] 10mm/sec FINE;
   1:  PR[GP1:91,1] = PR[GP1:90,1] + 129.938;
   1:  PR[GP1:91,2] = PR[GP1:90,2] + 108.788;
   1:L PR[91] 10mm/sec FINE;
   1:  PR[GP1:91,1] = PR[GP1:90,1] + 130.010;
   1:  PR[GP1:91,2] = PR[GP1:90,2] + 109.450;
   1:L PR[91] 10mm/sec FINE;
   1:  PR[GP1:91,1] = PR[GP1:90,1] + 129.608;
   1:  PR[GP1:91,2] = PR[GP1:90,2] + 112.864;
   1:L PR[91] 10mm/sec FINE;
   1:  PR[GP1:91,1] = PR[GP1:90,1] + 128.534;
   1:  PR[GP1:91,2] = PR[GP1:90,2] + 116.141;
   1:L PR[91] 10mm/sec FINE;
   1:  PR[GP1:91,1] = PR[GP1:90,1] + 126.790;
   1:  PR[GP1:91,2] = PR[GP1:90,2] + 119.145;
   1:L PR[91] 10mm/sec FINE;
   1:  PR[GP1:91,1] = PR[GP1:90,1] + 124.445;
   1:  PR[GP1:91,2] = PR[GP1:90,2] + 121.761;
   1:L PR[91] 10mm/sec FINE;
   1:  PR[GP1:91,1] = PR[GP1:90,1] + 122.375;
   1:  PR[GP1:91,2] = PR[GP1:90,2] + 123.303;
   1:L PR[91] 10mm/sec FINE;
   1:  PR[GP1:91,1] = PR[GP1:90,1] + 121.577;
   1:  PR[GP1:91,2] = PR[GP1:90,2] + 123.880;
   1:L PR[91] 10mm/sec FINE;
   1:  PR[GP1:91,1] = PR[GP1:90,1] + 118.256;
   1:  PR[GP1:91,2] = PR[GP1:90,2] + 125.412;
   1:L PR[91] 10mm/sec FINE;
   1:  PR[GP1:91,1] = PR[GP1:90,1] + 114.662;
   1:  PR[GP1:91,2] = PR[GP1:90,2] + 126.313;
   1:L PR[91] 10mm/sec FINE;
   1:  PR[GP1:91,1] = PR[GP1:90,1] + 110.911;
   1:  PR[GP1:91,2] = PR[GP1:90,2] + 126.522;
   1:L PR[91] 10mm/sec FINE;
   1:  PR[GP1:91,1] = PR[GP1:90,1] + 109.526;
   1:  PR[GP1:91,2] = PR[GP1:90,2] + 126.349;
   1:L PR[91] 10mm/sec FINE;
   1:  PR[GP1:91,1] = PR[GP1:90,1] + 107.163;
   1:  PR[GP1:91,2] = PR[GP1:90,2] + 126.047;
   1:L PR[91] 10mm/sec FINE;
   1:  PR[GP1:91,1] = PR[GP1:90,1] + 103.574;
   1:  PR[GP1:91,2] = PR[GP1:90,2] + 124.915;
   1:L PR[91] 10mm/sec FINE;
   1:  PR[GP1:91,1] = PR[GP1:90,1] + 100.281;
   1:  PR[GP1:91,2] = PR[GP1:90,2] + 123.161;
   1:L PR[91] 10mm/sec FINE;
   1:  PR[GP1:91,1] = PR[GP1:90,1] + 98.852;
   1:  PR[GP1:91,2] = PR[GP1:90,2] + 122.041;
   1:L PR[91] 10mm/sec FINE;
   1:  PR[GP1:91,1] = PR[GP1:90,1] + 97.399;
   1:  PR[GP1:91,2] = PR[GP1:90,2] + 120.860;
   1:L PR[91] 10mm/sec FINE;
   1:  PR[GP1:91,1] = PR[GP1:90,1] + 96.070;
   1:  PR[GP1:91,2] = PR[GP1:90,2] + 119.401;
   1:L PR[91] 10mm/sec FINE;
   1:  PR[GP1:91,1] = PR[GP1:90,1] + 95.584;
   1:  PR[GP1:91,2] = PR[GP1:90,2] + 119.116;
   1:L PR[91] 10mm/sec FINE;
   1:  PR[GP1:91,1] = PR[GP1:90,1] + 95.225;
   1:  PR[GP1:91,2] = PR[GP1:90,2] + 118.794;
   1:L PR[91] 10mm/sec FINE;
   1:  PR[GP1:91,1] = PR[GP1:90,1] + 94.965;
   1:  PR[GP1:91,2] = PR[GP1:90,2] + 118.743;
   1:L PR[91] 10mm/sec FINE;
   1:  PR[GP1:91,1] = PR[GP1:90,1] + 94.129;
   1:  PR[GP1:91,2] = PR[GP1:90,2] + 118.666;
   1:L PR[91] 10mm/sec FINE;
   1:  PR[GP1:91,1] = PR[GP1:90,1] + 93.635;
   1:  PR[GP1:91,2] = PR[GP1:90,2] + 118.907;
   1:L PR[91] 10mm/sec FINE;
   1:  PR[GP1:91,1] = PR[GP1:90,1] + 93.144;
   1:  PR[GP1:91,2] = PR[GP1:90,2] + 119.120;
   1:L PR[91] 10mm/sec FINE;
   1:  PR[GP1:91,1] = PR[GP1:90,1] + 92.873;
   1:  PR[GP1:91,2] = PR[GP1:90,2] + 119.398;
   1:L PR[91] 10mm/sec FINE;
   1:  PR[GP1:91,1] = PR[GP1:90,1] + 90.716;
   1:  PR[GP1:91,2] = PR[GP1:90,2] + 121.454;
   1:L PR[91] 10mm/sec FINE;
   1:  PR[GP1:91,1] = PR[GP1:90,1] + 89.793;
   1:  PR[GP1:91,2] = PR[GP1:90,2] + 122.251;
   1:L PR[91] 10mm/sec FINE;
   1:  PR[GP1:91,1] = PR[GP1:90,1] + 88.285;
   1:  PR[GP1:91,2] = PR[GP1:90,2] + 123.210;
   1:L PR[91] 10mm/sec FINE;
   1:  PR[GP1:91,1] = PR[GP1:90,1] + 86.259;
   1:  PR[GP1:91,2] = PR[GP1:90,2] + 124.379;
   1:L PR[91] 10mm/sec FINE;
   1:  PR[GP1:91,1] = PR[GP1:90,1] + 85.574;
   1:  PR[GP1:91,2] = PR[GP1:90,2] + 124.649;
   1:L PR[91] 10mm/sec FINE;
   1:  PR[GP1:91,1] = PR[GP1:90,1] + 82.490;
   1:  PR[GP1:91,2] = PR[GP1:90,2] + 125.736;
   1:L PR[91] 10mm/sec FINE;
   1:  PR[GP1:91,1] = PR[GP1:90,1] + 79.660;
   1:  PR[GP1:91,2] = PR[GP1:90,2] + 126.175;
   1:L PR[91] 10mm/sec FINE;
   1:  PR[GP1:91,1] = PR[GP1:90,1] + 78.804;
   1:  PR[GP1:91,2] = PR[GP1:90,2] + 126.295;
   1:L PR[91] 10mm/sec FINE;
   1:  PR[GP1:91,1] = PR[GP1:90,1] + 76.595;
   1:  PR[GP1:91,2] = PR[GP1:90,2] + 126.204;
   1:L PR[91] 10mm/sec FINE;
   1:  PR[GP1:91,1] = PR[GP1:90,1] + 75.124;
   1:  PR[GP1:91,2] = PR[GP1:90,2] + 126.125;
   1:L PR[91] 10mm/sec FINE;
   1:  PR[GP1:91,1] = PR[GP1:90,1] + 71.593;
   1:  PR[GP1:91,2] = PR[GP1:90,2] + 125.246;
   1:L PR[91] 10mm/sec FINE;
   1:  PR[GP1:91,1] = PR[GP1:90,1] + 68.350;
   1:  PR[GP1:91,2] = PR[GP1:90,2] + 123.706;
   1:L PR[91] 10mm/sec FINE;
   1:  PR[GP1:91,1] = PR[GP1:90,1] + 67.640;
   1:  PR[GP1:91,2] = PR[GP1:90,2] + 123.176;
   1:L PR[91] 10mm/sec FINE;
   1:  PR[GP1:91,1] = PR[GP1:90,1] + 65.520;
   1:  PR[GP1:91,2] = PR[GP1:90,2] + 121.571;
   1:L PR[91] 10mm/sec FINE;
   1:  PR[GP1:91,1] = PR[GP1:90,1] + 63.214;
   1:  PR[GP1:91,2] = PR[GP1:90,2] + 118.926;
   1:L PR[91] 10mm/sec FINE;
   1:  PR[GP1:91,1] = PR[GP1:90,1] + 61.512;
   1:  PR[GP1:91,2] = PR[GP1:90,2] + 115.882;
   1:L PR[91] 10mm/sec FINE;
   1:  PR[GP1:91,1] = PR[GP1:90,1] + 60.467;
   1:  PR[GP1:91,2] = PR[GP1:90,2] + 112.567;
   1:L PR[91] 10mm/sec FINE;
   1:  PR[GP1:91,1] = PR[GP1:90,1] + 60.166;
   1:  PR[GP1:91,2] = PR[GP1:90,2] + 109.088;
   1:L PR[91] 10mm/sec FINE;
   1:  PR[GP1:91,1] = PR[GP1:90,1] + 60.602;
   1:  PR[GP1:91,2] = PR[GP1:90,2] + 105.581;
   1:L PR[91] 10mm/sec FINE;
   1:  PR[GP1:91,1] = PR[GP1:90,1] + 61.727;
   1:  PR[GP1:91,2] = PR[GP1:90,2] + 102.213;
   1:L PR[91] 10mm/sec FINE;
   1:  PR[GP1:91,1] = PR[GP1:90,1] + 62.926;
   1:  PR[GP1:91,2] = PR[GP1:90,2] + 100.151;
   1:L PR[91] 10mm/sec FINE;
   1:  PR[GP1:91,1] = PR[GP1:90,1] + 63.558;
   1:  PR[GP1:91,2] = PR[GP1:90,2] + 99.095;
   1:L PR[91] 10mm/sec FINE;
   1:  PR[GP1:91,1] = PR[GP1:90,1] + 64.887;
   1:  PR[GP1:91,2] = PR[GP1:90,2] + 97.598;
   1:L PR[91] 10mm/sec FINE;
   1:  PR[GP1:91,1] = PR[GP1:90,1] + 66.022;
   1:  PR[GP1:91,2] = PR[GP1:90,2] + 96.359;
   1:L PR[91] 10mm/sec FINE;
   1:  PR[GP1:91,1] = PR[GP1:90,1] + 67.222;
   1:  PR[GP1:91,2] = PR[GP1:90,2] + 95.449;
   1:L PR[91] 10mm/sec FINE;
   1:  PR[GP1:91,1] = PR[GP1:90,1] + 69.025;
   1:  PR[GP1:91,2] = PR[GP1:90,2] + 94.134;
   1:L PR[91] 10mm/sec FINE;
   1:  PR[GP1:91,1] = PR[GP1:90,1] + 72.548;
   1:  PR[GP1:91,2] = PR[GP1:90,2] + 92.536;
   1:  PR[GP1:91,3] = PR[GP1:90,3] + 20.900;
   1:L PR[91] 10mm/sec FINE;
   1:  PR[GP1:91,1] = PR[GP1:90,1] + 72.987;
   1:  PR[GP1:91,2] = PR[GP1:90,2] + 92.355;
   1:L PR[91] 10mm/sec FINE;
   1:  PR[GP1:91,1] = PR[GP1:90,1] + 75.631;
   1:  PR[GP1:91,2] = PR[GP1:90,2] + 91.695;
   1:L PR[91] 10mm/sec FINE;
   1:  PR[GP1:91,1] = PR[GP1:90,1] + 77.071;
   1:  PR[GP1:91,2] = PR[GP1:90,2] + 91.405;
   1:L PR[91] 10mm/sec FINE;
   1:  PR[GP1:91,1] = PR[GP1:90,1] + 78.743;
   1:  PR[GP1:91,2] = PR[GP1:90,2] + 91.309;
   1:L PR[91] 10mm/sec FINE;
   1:  PR[GP1:91,1] = PR[GP1:90,1] + 81.362;
   1:  PR[GP1:91,2] = PR[GP1:90,2] + 91.299;
   1:L PR[91] 10mm/sec FINE;
   1:  PR[GP1:91,1] = PR[GP1:90,1] + 81.820;
   1:  PR[GP1:91,2] = PR[GP1:90,2] + 91.361;
   1:L PR[91] 10mm/sec FINE;
   1:  PR[GP1:91,1] = PR[GP1:90,1] + 82.980;
   1:  PR[GP1:91,2] = PR[GP1:90,2] + 91.590;
   1:L PR[91] 10mm/sec FINE;
   1:  PR[GP1:91,1] = PR[GP1:90,1] + 85.143;
   1:  PR[GP1:91,2] = PR[GP1:90,2] + 91.927;
   1:L PR[91] 10mm/sec FINE;
   1:  PR[GP1:91,1] = PR[GP1:90,1] + 86.171;
   1:  PR[GP1:91,2] = PR[GP1:90,2] + 92.220;
   1:L PR[91] 10mm/sec FINE;
   1:  PR[GP1:91,1] = PR[GP1:90,1] + 88.295;
   1:  PR[GP1:91,2] = PR[GP1:90,2] + 93.001;
   1:L PR[91] 10mm/sec FINE;
   1:  PR[GP1:91,1] = PR[GP1:90,1] + 90.594;
   1:  PR[GP1:91,2] = PR[GP1:90,2] + 94.170;
   1:L PR[91] 10mm/sec FINE;
   1:  PR[GP1:91,1] = PR[GP1:90,1] + 91.058;
   1:  PR[GP1:91,2] = PR[GP1:90,2] + 94.464;
   1:L PR[91] 10mm/sec FINE;
   1:  PR[GP1:91,1] = PR[GP1:90,1] + 91.967;
   1:  PR[GP1:91,2] = PR[GP1:90,2] + 95.203;
   1:L PR[91] 10mm/sec FINE;
   1:  PR[GP1:91,1] = PR[GP1:90,1] + 93.551;
   1:  PR[GP1:91,2] = PR[GP1:90,2] + 96.335;
   1:L PR[91] 10mm/sec FINE;
   1:  PR[GP1:91,1] = PR[GP1:90,1] + 94.188;
   1:  PR[GP1:91,2] = PR[GP1:90,2] + 96.698;
   1:L PR[91] 10mm/sec FINE;
   1:  PR[GP1:91,1] = PR[GP1:90,1] + 94.365;
   1:  PR[GP1:91,2] = PR[GP1:90,2] + 96.775;
   1:L PR[91] 10mm/sec FINE;
   1:  PR[GP1:91,1] = PR[GP1:90,1] + 94.561;
   1:  PR[GP1:91,2] = PR[GP1:90,2] + 96.788;
   1:L PR[91] 10mm/sec FINE;
   1:  PR[GP1:91,1] = PR[GP1:90,1] + 95.287;
   1:  PR[GP1:91,2] = PR[GP1:90,2] + 96.748;
   1:L PR[91] 10mm/sec FINE;
   1:  PR[GP1:91,1] = PR[GP1:90,1] + 95.497;
   1:  PR[GP1:91,2] = PR[GP1:90,2] + 96.689;
   1:L PR[91] 10mm/sec FINE;
   1:  PR[GP1:91,1] = PR[GP1:90,1] + 95.698;
   1:  PR[GP1:91,2] = PR[GP1:90,2] + 96.561;
   1:L PR[91] 10mm/sec FINE;
   1:  PR[GP1:91,1] = PR[GP1:90,1] + 95.929;
   1:  PR[GP1:91,2] = PR[GP1:90,2] + 96.365;
   1:L PR[91] 10mm/sec FINE;
   1:  PR[GP1:91,1] = PR[GP1:90,1] + 96.242;
   1:  PR[GP1:91,2] = PR[GP1:90,2] + 96.139;
   1:L PR[91] 10mm/sec FINE;
   1:  PR[GP1:91,1] = PR[GP1:90,1] + 96.876;
   1:  PR[GP1:91,2] = PR[GP1:90,2] + 95.573;
   1:L PR[91] 10mm/sec FINE;
   1:  PR[GP1:91,1] = PR[GP1:90,1] + 98.593;
   1:  PR[GP1:91,2] = PR[GP1:90,2] + 94.204;
   1:L PR[91] 10mm/sec FINE;
   1:  PR[GP1:91,1] = PR[GP1:90,1] + 99.262;
   1:  PR[GP1:91,2] = PR[GP1:90,2] + 93.790;
   1:L PR[91] 10mm/sec FINE;
   1:  PR[GP1:91,1] = PR[GP1:90,1] + 100.873;
   1:  PR[GP1:91,2] = PR[GP1:90,2] + 92.872;
   1:L PR[91] 10mm/sec FINE;
   1:  PR[GP1:91,1] = PR[GP1:90,1] + 102.025;
   1:  PR[GP1:91,2] = PR[GP1:90,2] + 92.388;
   1:L PR[91] 10mm/sec FINE;
   1:  PR[GP1:91,1] = PR[GP1:90,1] + 103.348;
   1:  PR[GP1:91,2] = PR[GP1:90,2] + 91.881;
   1:L PR[91] 10mm/sec FINE;
   1:  PR[GP1:91,1] = PR[GP1:90,1] + 105.178;
   1:  PR[GP1:91,2] = PR[GP1:90,2] + 91.422;
   1:L PR[91] 10mm/sec FINE;
   1:  PR[GP1:91,1] = PR[GP1:90,1] + 105.966;
   1:  PR[GP1:91,2] = PR[GP1:90,2] + 91.247;
   1:L PR[91] 10mm/sec FINE;
   1:  PR[GP1:91,1] = PR[GP1:90,1] + 108.681;
   1:  PR[GP1:91,2] = PR[GP1:90,2] + 90.984;
   1:L PR[91] 10mm/sec FINE;
   1:  PR[GP1:91,1] = PR[GP1:90,1] + 111.461;
   1:  PR[GP1:91,2] = PR[GP1:90,2] + 91.070;
   1:L PR[91] 10mm/sec FINE;
   1:  PR[GP1:91,1] = PR[GP1:90,1] + 112.546;
   1:  PR[GP1:91,2] = PR[GP1:90,2] + 91.234;
   1:L PR[91] 10mm/sec FINE;
   1:  PR[GP1:91,1] = PR[GP1:90,1] + 114.232;
   1:  PR[GP1:91,2] = PR[GP1:90,2] + 91.525;
   1:L PR[91] 10mm/sec FINE;
   1:  PR[GP1:91,1] = PR[GP1:90,1] + 116.945;
   1:  PR[GP1:91,2] = PR[GP1:90,2] + 92.351;
   1:L PR[91] 10mm/sec FINE;
   1:  PR[GP1:91,1] = PR[GP1:90,1] + 117.925;
   1:  PR[GP1:91,2] = PR[GP1:90,2] + 92.805;
   1:L PR[91] 10mm/sec FINE;
   1:  PR[GP1:91,1] = PR[GP1:90,1] + 119.563;
   1:  PR[GP1:91,2] = PR[GP1:90,2] + 93.529;
   1:L PR[91] 10mm/sec FINE;
   1:  PR[GP1:91,1] = PR[GP1:90,1] + 122.008;
   1:  PR[GP1:91,2] = PR[GP1:90,2] + 95.051;
   1:L PR[91] 10mm/sec FINE;
   1:  PR[GP1:91,1] = PR[GP1:90,1] + 124.210;
   1:  PR[GP1:91,2] = PR[GP1:90,2] + 96.899;
   1:L PR[91] 10mm/sec FINE;
   1:  PR[GP1:91,1] = PR[GP1:90,1] + 126.106;
   1:  PR[GP1:91,2] = PR[GP1:90,2] + 99.039;
   1:L PR[91] 10mm/sec FINE;
   1:  PR[GP1:91,1] = PR[GP1:90,1] + 127.620;
   1:  PR[GP1:91,2] = PR[GP1:90,2] + 101.427;
   1:L PR[91] 10mm/sec FINE;
   1:  PR[GP1:91,1] = PR[GP1:90,1] + 128.727;
   1:  PR[GP1:91,2] = PR[GP1:90,2] + 103.990;
   1:L PR[91] 10mm/sec FINE;
   1:  PR[GP1:91,1] = PR[GP1:90,1] + 129.399;
   1:  PR[GP1:91,2] = PR[GP1:90,2] + 106.668;
   1:L PR[91] 10mm/sec FINE;
   1:  PR[GP1:91,1] = PR[GP1:90,1] + 129.637;
   1:  PR[GP1:91,2] = PR[GP1:90,2] + 109.403;
   1:L PR[91] 10mm/sec FINE;
   1:  PR[GP1:91,1] = PR[GP1:90,1] + 129.488;
   1:  PR[GP1:91,2] = PR[GP1:90,2] + 110.807;
   1:L PR[91] 10mm/sec FINE;
   1:  PR[GP1:91,1] = PR[GP1:90,1] + 129.249;
   1:  PR[GP1:91,2] = PR[GP1:90,2] + 112.826;
   1:L PR[91] 10mm/sec FINE;
   1:  PR[GP1:91,1] = PR[GP1:90,1] + 128.169;
   1:  PR[GP1:91,2] = PR[GP1:90,2] + 116.105;
   1:L PR[91] 10mm/sec FINE;
   1:  PR[GP1:91,1] = PR[GP1:90,1] + 126.419;
   1:  PR[GP1:91,2] = PR[GP1:90,2] + 119.110;
   1:L PR[91] 10mm/sec FINE;
   1:  PR[GP1:91,1] = PR[GP1:90,1] + 124.985;
   1:  PR[GP1:91,2] = PR[GP1:90,2] + 120.707;
   1:L PR[91] 10mm/sec FINE;
   1:  PR[GP1:91,1] = PR[GP1:90,1] + 124.054;
   1:  PR[GP1:91,2] = PR[GP1:90,2] + 121.718;
   1:L PR[91] 10mm/sec FINE;
   1:  PR[GP1:91,1] = PR[GP1:90,1] + 121.139;
   1:  PR[GP1:91,2] = PR[GP1:90,2] + 123.825;
   1:L PR[91] 10mm/sec FINE;
   1:  PR[GP1:91,1] = PR[GP1:90,1] + 117.816;
   1:  PR[GP1:91,2] = PR[GP1:90,2] + 125.356;
   1:L PR[91] 10mm/sec FINE;
   1:  PR[GP1:91,1] = PR[GP1:90,1] + 115.907;
   1:  PR[GP1:91,2] = PR[GP1:90,2] + 125.835;
   1:L PR[91] 10mm/sec FINE;
   1:  PR[GP1:91,1] = PR[GP1:90,1] + 114.216;
   1:  PR[GP1:91,2] = PR[GP1:90,2] + 126.238;
   1:L PR[91] 10mm/sec FINE;
   1:  PR[GP1:91,1] = PR[GP1:90,1] + 110.466;
   1:  PR[GP1:91,2] = PR[GP1:90,2] + 126.437;
   1:L PR[91] 10mm/sec FINE;
   1:  PR[GP1:91,1] = PR[GP1:90,1] + 106.715;
   1:  PR[GP1:91,2] = PR[GP1:90,2] + 125.967;
   1:L PR[91] 10mm/sec FINE;
   1:  PR[GP1:91,1] = PR[GP1:90,1] + 103.154;
   1:  PR[GP1:91,2] = PR[GP1:90,2] + 124.816;
   1:L PR[91] 10mm/sec FINE;
   1:  PR[GP1:91,1] = PR[GP1:90,1] + 99.846;
   1:  PR[GP1:91,2] = PR[GP1:90,2] + 123.071;
   1:L PR[91] 10mm/sec FINE;
   1:  PR[GP1:91,1] = PR[GP1:90,1] + 96.994;
   1:  PR[GP1:91,2] = PR[GP1:90,2] + 120.755;
   1:L PR[91] 10mm/sec FINE;
   1:  PR[GP1:91,1] = PR[GP1:90,1] + 96.079;
   1:  PR[GP1:91,2] = PR[GP1:90,2] + 119.751;
   1:L PR[91] 10mm/sec FINE;
   1:  PR[GP1:91,1] = PR[GP1:90,1] + 95.166;
   1:  PR[GP1:91,2] = PR[GP1:90,2] + 119.209;
   1:L PR[91] 10mm/sec FINE;
   1:  PR[GP1:91,1] = PR[GP1:90,1] + 94.166;
   1:  PR[GP1:91,2] = PR[GP1:90,2] + 119.126;
   1:L PR[91] 10mm/sec FINE;
   1:  PR[GP1:91,1] = PR[GP1:90,1] + 94.088;
   1:  PR[GP1:91,2] = PR[GP1:90,2] + 119.127;
   1:L PR[91] 10mm/sec FINE;
   1:  PR[GP1:91,1] = PR[GP1:90,1] + 93.141;
   1:  PR[GP1:91,2] = PR[GP1:90,2] + 119.546;
   1:L PR[91] 10mm/sec FINE;
   1:  PR[GP1:91,1] = PR[GP1:90,1] + 92.968;
   1:  PR[GP1:91,2] = PR[GP1:90,2] + 119.723;
   1:L PR[91] 10mm/sec FINE;
   1:  PR[GP1:91,1] = PR[GP1:90,1] + 91.346;
   1:  PR[GP1:91,2] = PR[GP1:90,2] + 121.132;
   1:L PR[91] 10mm/sec FINE;
   1:  PR[GP1:91,1] = PR[GP1:90,1] + 90.688;
   1:  PR[GP1:91,2] = PR[GP1:90,2] + 121.763;
   1:L PR[91] 10mm/sec FINE;
   1:  PR[GP1:91,1] = PR[GP1:90,1] + 90.399;
   1:  PR[GP1:91,2] = PR[GP1:90,2] + 122.012;
   1:L PR[91] 10mm/sec FINE;
   1:  PR[GP1:91,1] = PR[GP1:90,1] + 88.213;
   1:  PR[GP1:91,2] = PR[GP1:90,2] + 123.404;
   1:L PR[91] 10mm/sec FINE;
   1:  PR[GP1:91,1] = PR[GP1:90,1] + 86.850;
   1:  PR[GP1:91,2] = PR[GP1:90,2] + 124.190;
   1:L PR[91] 10mm/sec FINE;
   1:  PR[GP1:91,1] = PR[GP1:90,1] + 85.478;
   1:  PR[GP1:91,2] = PR[GP1:90,2] + 124.731;
   1:L PR[91] 10mm/sec FINE;
   1:  PR[GP1:91,1] = PR[GP1:90,1] + 83.004;
   1:  PR[GP1:91,2] = PR[GP1:90,2] + 125.600;
   1:L PR[91] 10mm/sec FINE;
   1:  PR[GP1:91,1] = PR[GP1:90,1] + 82.513;
   1:  PR[GP1:91,2] = PR[GP1:90,2] + 125.692;
   1:L PR[91] 10mm/sec FINE;
   1:  PR[GP1:91,1] = PR[GP1:90,1] + 79.148;
   1:  PR[GP1:91,2] = PR[GP1:90,2] + 126.208;
   1:L PR[91] 10mm/sec FINE;
   1:  PR[GP1:91,1] = PR[GP1:90,1] + 75.456;
   1:  PR[GP1:91,2] = PR[GP1:90,2] + 126.045;
   1:L PR[91] 10mm/sec FINE;
   1:  PR[GP1:91,1] = PR[GP1:90,1] + 71.917;
   1:  PR[GP1:91,2] = PR[GP1:90,2] + 125.170;
   1:L PR[91] 10mm/sec FINE;
   1:  PR[GP1:91,1] = PR[GP1:90,1] + 68.664;
   1:  PR[GP1:91,2] = PR[GP1:90,2] + 123.630;
   1:L PR[91] 10mm/sec FINE;
   1:  PR[GP1:91,1] = PR[GP1:90,1] + 67.552;
   1:  PR[GP1:91,2] = PR[GP1:90,2] + 122.799;
   1:L PR[91] 10mm/sec FINE;
   1:  PR[GP1:91,1] = PR[GP1:90,1] + 65.826;
   1:  PR[GP1:91,2] = PR[GP1:90,2] + 121.493;
   1:L PR[91] 10mm/sec FINE;
   1:  PR[GP1:91,1] = PR[GP1:90,1] + 63.515;
   1:  PR[GP1:91,2] = PR[GP1:90,2] + 118.845;
   1:L PR[91] 10mm/sec FINE;
   1:  PR[GP1:91,1] = PR[GP1:90,1] + 61.809;
   1:  PR[GP1:91,2] = PR[GP1:90,2] + 115.796;
   1:L PR[91] 10mm/sec FINE;
   1:  PR[GP1:91,1] = PR[GP1:90,1] + 60.761;
   1:  PR[GP1:91,2] = PR[GP1:90,2] + 112.476;
   1:L PR[91] 10mm/sec FINE;
   1:  PR[GP1:91,1] = PR[GP1:90,1] + 60.458;
   1:  PR[GP1:91,2] = PR[GP1:90,2] + 108.990;
   1:L PR[91] 10mm/sec FINE;
   1:  PR[GP1:91,1] = PR[GP1:90,1] + 60.740;
   1:  PR[GP1:91,2] = PR[GP1:90,2] + 106.669;
   1:L PR[91] 10mm/sec FINE;
   1:  PR[GP1:91,1] = PR[GP1:90,1] + 60.903;
   1:  PR[GP1:91,2] = PR[GP1:90,2] + 105.473;
   1:L PR[91] 10mm/sec FINE;
   1:  PR[GP1:91,1] = PR[GP1:90,1] + 62.033;
   1:  PR[GP1:91,2] = PR[GP1:90,2] + 102.097;
   1:L PR[91] 10mm/sec FINE;
   1:  PR[GP1:91,1] = PR[GP1:90,1] + 62.978;
   1:  PR[GP1:91,2] = PR[GP1:90,2] + 100.473;
   1:L PR[91] 10mm/sec FINE;
   1:  PR[GP1:91,1] = PR[GP1:90,1] + 63.876;
   1:  PR[GP1:91,2] = PR[GP1:90,2] + 98.970;
   1:L PR[91] 10mm/sec FINE;
   1:  PR[GP1:91,1] = PR[GP1:90,1] + 64.854;
   1:  PR[GP1:91,2] = PR[GP1:90,2] + 97.869;
   1:L PR[91] 10mm/sec FINE;
   1:  PR[GP1:91,1] = PR[GP1:90,1] + 66.357;
   1:  PR[GP1:91,2] = PR[GP1:90,2] + 96.230;
   1:L PR[91] 10mm/sec FINE;
   1:  PR[GP1:91,1] = PR[GP1:90,1] + 67.113;
   1:  PR[GP1:91,2] = PR[GP1:90,2] + 95.656;
   1:L PR[91] 10mm/sec FINE;
   1:  PR[GP1:91,1] = PR[GP1:90,1] + 69.378;
   1:  PR[GP1:91,2] = PR[GP1:90,2] + 94.004;
   1:L PR[91] 10mm/sec FINE;
   1:  PR[GP1:91,1] = PR[GP1:90,1] + 72.500;
   1:  PR[GP1:91,2] = PR[GP1:90,2] + 92.610;
   1:  PR[GP1:91,3] = PR[GP1:90,3] + 21.900;
   1:L PR[91] 10mm/sec FINE;
   1:  PR[GP1:91,1] = PR[GP1:90,1] + 73.567;
   1:  PR[GP1:91,2] = PR[GP1:90,2] + 92.169;
   1:L PR[91] 10mm/sec FINE;
   1:  PR[GP1:91,1] = PR[GP1:90,1] + 75.534;
   1:  PR[GP1:91,2] = PR[GP1:90,2] + 91.678;
   1:L PR[91] 10mm/sec FINE;
   1:  PR[GP1:91,1] = PR[GP1:90,1] + 77.702;
   1:  PR[GP1:91,2] = PR[GP1:90,2] + 91.241;
   1:L PR[91] 10mm/sec FINE;
   1:  PR[GP1:91,1] = PR[GP1:90,1] + 78.611;
   1:  PR[GP1:91,2] = PR[GP1:90,2] + 91.190;
   1:L PR[91] 10mm/sec FINE;
   1:  PR[GP1:91,1] = PR[GP1:90,1] + 80.911;
   1:  PR[GP1:91,2] = PR[GP1:90,2] + 91.181;
   1:L PR[91] 10mm/sec FINE;
   1:  PR[GP1:91,1] = PR[GP1:90,1] + 81.858;
   1:  PR[GP1:91,2] = PR[GP1:90,2] + 91.149;
   1:L PR[91] 10mm/sec FINE;
   1:  PR[GP1:91,1] = PR[GP1:90,1] + 82.335;
   1:  PR[GP1:91,2] = PR[GP1:90,2] + 91.194;
   1:L PR[91] 10mm/sec FINE;
   1:  PR[GP1:91,1] = PR[GP1:90,1] + 85.318;
   1:  PR[GP1:91,2] = PR[GP1:90,2] + 91.658;
   1:L PR[91] 10mm/sec FINE;
   1:  PR[GP1:91,1] = PR[GP1:90,1] + 87.477;
   1:  PR[GP1:91,2] = PR[GP1:90,2] + 92.274;
   1:L PR[91] 10mm/sec FINE;
   1:  PR[GP1:91,1] = PR[GP1:90,1] + 88.430;
   1:  PR[GP1:91,2] = PR[GP1:90,2] + 92.624;
   1:L PR[91] 10mm/sec FINE;
   1:  PR[GP1:91,1] = PR[GP1:90,1] + 90.110;
   1:  PR[GP1:91,2] = PR[GP1:90,2] + 93.479;
   1:L PR[91] 10mm/sec FINE;
   1:  PR[GP1:91,1] = PR[GP1:90,1] + 91.331;
   1:  PR[GP1:91,2] = PR[GP1:90,2] + 94.013;
   1:L PR[91] 10mm/sec FINE;
   1:  PR[GP1:91,1] = PR[GP1:90,1] + 91.809;
   1:  PR[GP1:91,2] = PR[GP1:90,2] + 94.290;
   1:L PR[91] 10mm/sec FINE;
   1:  PR[GP1:91,1] = PR[GP1:90,1] + 93.789;
   1:  PR[GP1:91,2] = PR[GP1:90,2] + 95.706;
   1:L PR[91] 10mm/sec FINE;
   1:  PR[GP1:91,1] = PR[GP1:90,1] + 94.215;
   1:  PR[GP1:91,2] = PR[GP1:90,2] + 95.948;
   1:L PR[91] 10mm/sec FINE;
   1:  PR[GP1:91,1] = PR[GP1:90,1] + 94.523;
   1:  PR[GP1:91,2] = PR[GP1:90,2] + 96.082;
   1:L PR[91] 10mm/sec FINE;
   1:  PR[GP1:91,1] = PR[GP1:90,1] + 94.862;
   1:  PR[GP1:91,2] = PR[GP1:90,2] + 96.104;
   1:L PR[91] 10mm/sec FINE;
   1:  PR[GP1:91,1] = PR[GP1:90,1] + 95.349;
   1:  PR[GP1:91,2] = PR[GP1:90,2] + 96.077;
   1:L PR[91] 10mm/sec FINE;
   1:  PR[GP1:91,1] = PR[GP1:90,1] + 95.701;
   1:  PR[GP1:91,2] = PR[GP1:90,2] + 95.980;
   1:L PR[91] 10mm/sec FINE;
   1:  PR[GP1:91,1] = PR[GP1:90,1] + 96.047;
   1:  PR[GP1:91,2] = PR[GP1:90,2] + 95.759;
   1:L PR[91] 10mm/sec FINE;
   1:  PR[GP1:91,1] = PR[GP1:90,1] + 96.363;
   1:  PR[GP1:91,2] = PR[GP1:90,2] + 95.490;
   1:L PR[91] 10mm/sec FINE;
   1:  PR[GP1:91,1] = PR[GP1:90,1] + 98.323;
   1:  PR[GP1:91,2] = PR[GP1:90,2] + 93.936;
   1:L PR[91] 10mm/sec FINE;
   1:  PR[GP1:91,1] = PR[GP1:90,1] + 100.618;
   1:  PR[GP1:91,2] = PR[GP1:90,2] + 92.624;
   1:L PR[91] 10mm/sec FINE;
   1:  PR[GP1:91,1] = PR[GP1:90,1] + 101.076;
   1:  PR[GP1:91,2] = PR[GP1:90,2] + 92.432;
   1:L PR[91] 10mm/sec FINE;
   1:  PR[GP1:91,1] = PR[GP1:90,1] + 103.101;
   1:  PR[GP1:91,2] = PR[GP1:90,2] + 91.655;
   1:L PR[91] 10mm/sec FINE;
   1:  PR[GP1:91,1] = PR[GP1:90,1] + 104.137;
   1:  PR[GP1:91,2] = PR[GP1:90,2] + 91.396;
   1:L PR[91] 10mm/sec FINE;
   1:  PR[GP1:91,1] = PR[GP1:90,1] + 105.723;
   1:  PR[GP1:91,2] = PR[GP1:90,2] + 91.044;
   1:L PR[91] 10mm/sec FINE;
   1:  PR[GP1:91,1] = PR[GP1:90,1] + 107.544;
   1:  PR[GP1:91,2] = PR[GP1:90,2] + 90.867;
   1:L PR[91] 10mm/sec FINE;
   1:  PR[GP1:91,1] = PR[GP1:90,1] + 108.433;
   1:  PR[GP1:91,2] = PR[GP1:90,2] + 90.802;
   1:L PR[91] 10mm/sec FINE;
   1:  PR[GP1:91,1] = PR[GP1:90,1] + 111.184;
   1:  PR[GP1:91,2] = PR[GP1:90,2] + 90.935;
   1:L PR[91] 10mm/sec FINE;
   1:  PR[GP1:91,1] = PR[GP1:90,1] + 113.948;
   1:  PR[GP1:91,2] = PR[GP1:90,2] + 91.411;
   1:L PR[91] 10mm/sec FINE;
   1:  PR[GP1:91,1] = PR[GP1:90,1] + 115.139;
   1:  PR[GP1:91,2] = PR[GP1:90,2] + 91.770;
   1:L PR[91] 10mm/sec FINE;
   1:  PR[GP1:91,1] = PR[GP1:90,1] + 116.646;
   1:  PR[GP1:91,2] = PR[GP1:90,2] + 92.253;
   1:L PR[91] 10mm/sec FINE;
   1:  PR[GP1:91,1] = PR[GP1:90,1] + 118.949;
   1:  PR[GP1:91,2] = PR[GP1:90,2] + 93.320;
   1:L PR[91] 10mm/sec FINE;
   1:  PR[GP1:91,1] = PR[GP1:90,1] + 119.227;
   1:  PR[GP1:91,2] = PR[GP1:90,2] + 93.455;
   1:L PR[91] 10mm/sec FINE;
   1:  PR[GP1:91,1] = PR[GP1:90,1] + 121.653;
   1:  PR[GP1:91,2] = PR[GP1:90,2] + 94.990;
   1:L PR[91] 10mm/sec FINE;
   1:  PR[GP1:91,1] = PR[GP1:90,1] + 123.840;
   1:  PR[GP1:91,2] = PR[GP1:90,2] + 96.843;
   1:L PR[91] 10mm/sec FINE;
   1:  PR[GP1:91,1] = PR[GP1:90,1] + 125.723;
   1:  PR[GP1:91,2] = PR[GP1:90,2] + 98.984;
   1:L PR[91] 10mm/sec FINE;
   1:  PR[GP1:91,1] = PR[GP1:90,1] + 127.250;
   1:  PR[GP1:91,2] = PR[GP1:90,2] + 101.368;
   1:L PR[91] 10mm/sec FINE;
   1:  PR[GP1:91,1] = PR[GP1:90,1] + 127.627;
   1:  PR[GP1:91,2] = PR[GP1:90,2] + 102.228;
   1:L PR[91] 10mm/sec FINE;
   1:  PR[GP1:91,1] = PR[GP1:90,1] + 128.361;
   1:  PR[GP1:91,2] = PR[GP1:90,2] + 103.934;
   1:L PR[91] 10mm/sec FINE;
   1:  PR[GP1:91,1] = PR[GP1:90,1] + 129.031;
   1:  PR[GP1:91,2] = PR[GP1:90,2] + 106.617;
   1:L PR[91] 10mm/sec FINE;
   1:  PR[GP1:91,1] = PR[GP1:90,1] + 129.255;
   1:  PR[GP1:91,2] = PR[GP1:90,2] + 109.354;
   1:L PR[91] 10mm/sec FINE;
   1:  PR[GP1:91,1] = PR[GP1:90,1] + 128.889;
   1:  PR[GP1:91,2] = PR[GP1:90,2] + 112.790;
   1:L PR[91] 10mm/sec FINE;
   1:  PR[GP1:91,1] = PR[GP1:90,1] + 127.799;
   1:  PR[GP1:91,2] = PR[GP1:90,2] + 116.066;
   1:L PR[91] 10mm/sec FINE;
   1:  PR[GP1:91,1] = PR[GP1:90,1] + 126.018;
   1:  PR[GP1:91,2] = PR[GP1:90,2] + 119.062;
   1:L PR[91] 10mm/sec FINE;
   1:  PR[GP1:91,1] = PR[GP1:90,1] + 123.620;
   1:  PR[GP1:91,2] = PR[GP1:90,2] + 121.664;
   1:L PR[91] 10mm/sec FINE;
   1:  PR[GP1:91,1] = PR[GP1:90,1] + 120.702;
   1:  PR[GP1:91,2] = PR[GP1:90,2] + 123.769;
   1:L PR[91] 10mm/sec FINE;
   1:  PR[GP1:91,1] = PR[GP1:90,1] + 117.378;
   1:  PR[GP1:91,2] = PR[GP1:90,2] + 125.298;
   1:L PR[91] 10mm/sec FINE;
   1:  PR[GP1:91,1] = PR[GP1:90,1] + 113.766;
   1:  PR[GP1:91,2] = PR[GP1:90,2] + 126.159;
   1:L PR[91] 10mm/sec FINE;
   1:  PR[GP1:91,1] = PR[GP1:90,1] + 112.186;
   1:  PR[GP1:91,2] = PR[GP1:90,2] + 126.246;
   1:L PR[91] 10mm/sec FINE;
   1:  PR[GP1:91,1] = PR[GP1:90,1] + 110.021;
   1:  PR[GP1:91,2] = PR[GP1:90,2] + 126.353;
   1:L PR[91] 10mm/sec FINE;
   1:  PR[GP1:91,1] = PR[GP1:90,1] + 107.886;
   1:  PR[GP1:91,2] = PR[GP1:90,2] + 126.086;
   1:L PR[91] 10mm/sec FINE;
   1:  PR[GP1:91,1] = PR[GP1:90,1] + 106.297;
   1:  PR[GP1:91,2] = PR[GP1:90,2] + 125.867;
   1:L PR[91] 10mm/sec FINE;
   1:  PR[GP1:91,1] = PR[GP1:90,1] + 102.735;
   1:  PR[GP1:91,2] = PR[GP1:90,2] + 124.717;
   1:L PR[91] 10mm/sec FINE;
   1:  PR[GP1:91,1] = PR[GP1:90,1] + 100.592;
   1:  PR[GP1:91,2] = PR[GP1:90,2] + 123.587;
   1:L PR[91] 10mm/sec FINE;
   1:  PR[GP1:91,1] = PR[GP1:90,1] + 99.458;
   1:  PR[GP1:91,2] = PR[GP1:90,2] + 122.962;
   1:L PR[91] 10mm/sec FINE;
   1:  PR[GP1:91,1] = PR[GP1:90,1] + 96.588;
   1:  PR[GP1:91,2] = PR[GP1:90,2] + 120.650;
   1:L PR[91] 10mm/sec FINE;
   1:  PR[GP1:91,1] = PR[GP1:90,1] + 96.088;
   1:  PR[GP1:91,2] = PR[GP1:90,2] + 120.101;
   1:L PR[91] 10mm/sec FINE;
   1:  PR[GP1:91,1] = PR[GP1:90,1] + 95.641;
   1:  PR[GP1:91,2] = PR[GP1:90,2] + 119.839;
   1:L PR[91] 10mm/sec FINE;
   1:  PR[GP1:91,1] = PR[GP1:90,1] + 95.196;
   1:  PR[GP1:91,2] = PR[GP1:90,2] + 119.533;
   1:L PR[91] 10mm/sec FINE;
   1:  PR[GP1:91,1] = PR[GP1:90,1] + 94.420;
   1:  PR[GP1:91,2] = PR[GP1:90,2] + 119.469;
   1:L PR[91] 10mm/sec FINE;
   1:  PR[GP1:91,1] = PR[GP1:90,1] + 94.101;
   1:  PR[GP1:91,2] = PR[GP1:90,2] + 119.472;
   1:L PR[91] 10mm/sec FINE;
   1:  PR[GP1:91,1] = PR[GP1:90,1] + 93.468;
   1:  PR[GP1:91,2] = PR[GP1:90,2] + 119.828;
   1:L PR[91] 10mm/sec FINE;
   1:  PR[GP1:91,1] = PR[GP1:90,1] + 93.147;
   1:  PR[GP1:91,2] = PR[GP1:90,2] + 119.967;
   1:L PR[91] 10mm/sec FINE;
   1:  PR[GP1:91,1] = PR[GP1:90,1] + 91.145;
   1:  PR[GP1:91,2] = PR[GP1:90,2] + 121.707;
   1:L PR[91] 10mm/sec FINE;
   1:  PR[GP1:91,1] = PR[GP1:90,1] + 90.753;
   1:  PR[GP1:91,2] = PR[GP1:90,2] + 121.977;
   1:L PR[91] 10mm/sec FINE;
   1:  PR[GP1:91,1] = PR[GP1:90,1] + 89.847;
   1:  PR[GP1:91,2] = PR[GP1:90,2] + 122.511;
   1:L PR[91] 10mm/sec FINE;
   1:  PR[GP1:91,1] = PR[GP1:90,1] + 88.141;
   1:  PR[GP1:91,2] = PR[GP1:90,2] + 123.598;
   1:L PR[91] 10mm/sec FINE;
   1:  PR[GP1:91,1] = PR[GP1:90,1] + 87.440;
   1:  PR[GP1:91,2] = PR[GP1:90,2] + 124.002;
   1:L PR[91] 10mm/sec FINE;
   1:  PR[GP1:91,1] = PR[GP1:90,1] + 85.382;
   1:  PR[GP1:91,2] = PR[GP1:90,2] + 124.813;
   1:L PR[91] 10mm/sec FINE;
   1:  PR[GP1:91,1] = PR[GP1:90,1] + 83.570;
   1:  PR[GP1:91,2] = PR[GP1:90,2] + 125.449;
   1:L PR[91] 10mm/sec FINE;
